VAR_INST
    {attribute 'hide'}
    bEncError           : BOOL;
END_VAR
// Save Encoder position
// needs some pre-conditions to use persistent storage
IF Enable THEN
    // Check ST_MotionStage for an encoder error (range 0x44nn)
    bEncError:=  stMotionStage.Axis.Status.Error AND  (  stMotionStage.Axis.Status.ErrorID  >= 16#4400  AND  stMotionStage.Axis.Status.ErrorID <= 16#44FF );
    // Do not save if we're currently loading or if there is an encoder error
    IF NOT bRestoreLoad AND NOT bEncError AND NOT bRestoreWaitRetry THEN
        fSavedPosition :=  stMotionStage.Axis.NcToPlc.ActPos;
        // This persistent variable lets us check if anything was saved
        // It will be TRUE at startup if we have saved values
        bSaved := TRUE;
    END_IF
END_IF
END_METHOD

{attribute 'call_after_init'}
(*  eModule: Mandatory must be unique for each MCS2 axis
    clears startup errors or warnings. the process is completed at run time
    SDO update of Drive and open Loop parameter Indexes based on module number
*)
METHOD PostInit
(* SDO update of Drive and open Loop parameter Indexes based on module number *)
stChanParams.nChanErrorCodeIdx        	:= nChanErrorCodeBase         	+ ((eModule-1) * nChanOfsBase);
stChanParams.nChanFErrWinIdx          	:= nChanFErrWinBase           	+ ((eModule-1) * nChanOfsBase);
stChanParams.nChanSoftLimitIdx        	:= nChanSoftLimitBase     		+ ((eModule-1) * nChanOfsBase);
stChanParams.nChanHomeOffsIdx         	:= nChanHomeOffsetBase        	+ ((eModule-1) * nChanOfsBase);
stChanParams.nChanHomeMethodIdx         := nChanHomeMethodBase       	+ ((eModule-1) * nChanOfsBase);
stChanParams.nChanHomeVeloIdx         	:= nChanHomingSpeedBase       	+ ((eModule-1) * nChanOfsBase);
stChanParams.nChanhomeAccIdx          	:= nChanhomingAccBase         	+ ((eModule-1) * nChanOfsBase);
stChanParams.nChanStepIdx             	:= nChanOlStepBase            	+ ((eModule-1) * nChanOfsBase);
stChanParams.nChanStepFreqIdx         	:= nChanOlStepFreqBase        	+ ((eModule-1) * nChanOfsBase);
stChanParams.nChanStepAmpIdx          	:= nChanOlStepAmpBase         	+ ((eModule-1) * nChanOfsBase);
stChanParams.nChanMaxCloseLoopFreqIdx   := nChanMaxCloseLoopFreqBase  	+ ((eModule-1) * nChanOfsBase);
stChanParams.nChanPositionerTypeIdx     := nChanPositionerTypeBase    	+ ((eModule-1) * nChanOfsBase);
stChanParams.nChanCalibrationOptIdx     := nCHanCalibrationOptBase    	+ ((eModule-1) * nChanOfsBase);
stChanParams.nChanSensorPowerModeIdx    := nChanSensorPowerModeBase   	+ ((eModule-1) * nChanOfsBase);
stChanParams.nChanReferencingOptIdx     := nChanReferencingOptBase    	+ ((eModule-1) * nChanOfsBase);
stChanParams.nChanReferenceTypeIdx      := nChanReferenceTypeBase     	+ ((eModule-1) * nChanOfsBase);
stChanParams.nChanSafeDirIdx            := nChanSafeDirBase           	+ ((eModule-1) * nChanOfsBase);
stChanParams.nChanMotorLoadIdx          := nChanMotorLoadBase         	+ ((eModule-1) * nChanOfsBase);
stChanParams.nChannelTypeIdx          	:= nChannelTypeBase       		+ ((eModule-1) * nChanOfsBase);
stChanParams.nChanStateIdx         		:= nChannelStateBase      		+ ((eModule-1) * nChanOfsBase);
stChanParams.nChanLogicalScaleOfsIdx   	:= nChanLogicalScaleOffsetBase	+ ((eModule-1) * nChanOfsBase);
stChanParams.nChanLogicalScaleInvIdx    := nChanLogicalScaleInvBase   	+ ((eModule-1) * nChanOfsBase);
stChanParams.nChanChannelTempIdx        := nChanChannelTempBase       	+ ((eModule-1) * nChanOfsBase);
stChanParams.nChanMovementTypeIdx       := nChanMovementTypeBase      	+ ((eModule-1) * nChanOfsBase);
stChanParams.nChanBaseUnitIdx           := nChanBaseUnitBase          	+ ((eModule-1) * nChanOfsBase);
stChanParams.nChanBaseResolutionIdx     := nChanBaseResolutionBase    	+ ((eModule-1) * nChanOfsBase);
stChanParams.nChanDistCodeInvIdx        := nChanDistCodeInvBase       	+ ((eModule-1) * nChanOfsBase);
stChanParams.nChanPositionerCtrlOptIdx  := nChanPositionerCtrlOptBase 	+ ((eModule-1) * nChanOfsBase);
stChanParams.nChanActuatorModeIdx       := nChanActuatorModeBase      	+ ((eModule-1) * nChanOfsBase);
stChanParams.nChanMotorLoadProtIdx      := nChanMotorLoadProtBase     	+ ((eModule-1) * nChanOfsBase);
stChanParams.nChanDiagClfIdx            := nChanDiagClfBase           	+ ((eModule-1) * nChanOfsBase);
bSystemInit := TRUE;
END_METHOD

METHOD PRIVATE PostMoveChecks : BOOL
VAR_INST
    rtAbortedHome        : R_TRIG;
    rtAbortedStepMove    : R_TRIG;
    rtAbortedCalibration : R_TRIG;
    rtResetDone          : R_TRIG;
    rtHaltDone           : R_TRIG;
    rtMoveDone           : R_TRIG;
    rtHomeDone           : R_TRIG;
    rtStepMoveDone       : R_TRIG;
    rtCalibrationDone    : R_TRIG;
    ftEnableFallEdge     : F_TRIG;
END_VAR
rtAbortedHome(CLK := fbhome.bHomeMoveAborted);
rtAbortedStepMove(CLK := fbStepMode.bStepMoveAborted);
rtAbortedCalibration(CLK := fbCalibrate.bCalibrateMoveAborted);

rtResetDone(CLK := fbMcReset.Done);
rtHaltDone(CLK := fbMcHalt.Done);

rtMoveDone(CLK := fbMcMoveAbsolute.Done);
rtHomeDone(CLK := fbhome.bHomeMoveDone);
rtStepMoveDone(CLK := fbStepMode.bStepMoveDone);
rtCalibrationDone(CLK := fbCalibrate.bCalibrateMoveDone);

IF rtAbortedHome.Q OR rtAbortedStepMove.Q OR rtAbortedCalibration.Q
   OR rtResetDone.Q OR rtHaltDone.Q
   OR rtMoveDone.Q OR rtHomeDone.Q OR rtStepMoveDone.Q OR rtCalibrationDone.Q THEN

    IF NOT stMotionStage.bDone THEN
        stMotionStage.bExecute := FALSE;;
        stMotionStage.bHomed := fbhome.bHomeMoveDone;
        IF rtMoveDone.Q THEN
            stMotionStage.bDone := TRUE;
            eDoneCause := E_MoveDoneCause.MoveDone;
        ELSIF rtStepMoveDone.Q THEN
            stMotionStage.bDone := TRUE;
            eDoneCause := E_MoveDoneCause.StepMoveDone;
        ELSIF rtHomeDone.Q THEN
            stMotionStage.bDone := TRUE;
            eDoneCause := E_MoveDoneCause.HomeDone;
            // Homing runs in DS402 manual HOME mode. Request closed-loop so the
            // drive manager switches the drive back to CSP now that homing is done.
            stChanParams.eOpModeReq := E_MCS2OpModeReq.CLOSED_LOOP;
        ELSIF rtCalibrationDone.Q THEN
            stMotionStage.bDone := TRUE;
            eDoneCause := E_MoveDoneCause.CalibrationDone;
            // Calibration runs in DS402 manual CALIBRATE mode. Request closed-loop so
            // the drive manager switches the drive back to CSP now that calibration is done.
            stChanParams.eOpModeReq := E_MCS2OpModeReq.CLOSED_LOOP;
        ELSIF rtResetDone.Q THEN
            stMotionStage.bDone := TRUE;
            eDoneCause := E_MoveDoneCause.ResetDone;
        ELSIF rtHaltDone.Q THEN
            stMotionStage.bDone := TRUE;
            eDoneCause := E_MoveDoneCause.HaltDone;
        ELSIF rtAbortedHome.Q THEN
            stMotionStage.bDone := TRUE;
            eDoneCause := E_MoveDoneCause.AbortedHome;
        ELSIF rtAbortedStepMove.Q THEN
            stMotionStage.bDone := TRUE;
            eDoneCause := E_MoveDoneCause.AbortedStepMove;
        ELSIF rtAbortedCalibration.Q THEN
            stMotionStage.bDone := TRUE;
            eDoneCause := E_MoveDoneCause.AbortedCalibration;
        END_IF
        IF rtHomeDone.Q OR rtAbortedHome.Q OR rtCalibrationDone.Q OR rtAbortedCalibration.Q THEN
            bEnPosLag       := bRecentEnPosLagStatus;
            fParameterValue := BOOL_TO_LREAL(bRecentEnPosLagStatus);
        END_IF
        IF fbDriveManager.bDS402Manual
           AND NOT (rtHomeDone.Q OR rtAbortedHome.Q OR rtCalibrationDone.Q OR rtAbortedCalibration.Q) THEN
            bEnPosLag := FALSE;
        END_IF
        IF (stMotionStage.nEnableMode = E_StageEnableMode.DURING_MOTION) THEN
            bPositionHold := TRUE;
            tonHoldTime.IN := TRUE;
        END_IF
        // get stable current position storage
        stChanParams.fPosition := stMotionStage.fPosition;
    END_IF
END_IF

tonHoldTime(PT := UDINT_TO_TIME(stChanParams.nHoldTime));
IF tonHoldTime.Q THEN
    bPositionHold := FALSE;
    tonHoldTime.IN := FALSE;
    bLastHoltTimeOut := TRUE;
END_IF

(* updated axis status
   Not needed in manual mode *)
IF NOT fbDriveManager.bDS402Manual THEN
     stMotionStage.Axis.ReadStatus();
END_IF

bPrepareDisable S= (stMotionStage.nEnableMode = E_StageEnableMode.DURING_MOTION) AND ftExec.Q;

IF bPrepareDisable AND fbDriveManager.bCSPModeEnabled THEN
    IF stMotionStage.Axis.Status.StandStill THEN
        IF NOT bPositionHold THEN
            bPrepareDisable := FALSE;
            stMotionStage.bEnable := FALSE; // TwinCAT NC disables MC_Power (CSP)
        END_IF
    END_IF
ELSIF bPrepareDisable AND fbDriveManager.bDS402Manual THEN
    IF fbDriveManager.bOperational THEN
        IF NOT bPositionHold THEN
            bPrepareDisable := FALSE;
            stMotionStage.bEnable := FALSE; // Manual disables via drive control word
        END_IF
    END_IF
END_IF

ftEnableFallEdge(CLK := stMotionStage.bEnable);
IF ftEnableFallEdge.Q THEN
    // Only power off in manual if we're staying in manual. During a switch back
    // to CSP, let the NC ramp the control word down so it isn't disabled under it.
    IF fbDriveManager.bDS402Manual
       AND stChanParams.eOpModeReq <> E_MCS2OpModeReq.CLOSED_LOOP THEN
        stDS402Drive.nDriveControl := 6; // Manual mode power off
    END_IF
END_IF
END_METHOD

METHOD Power
fbMcPower(
    Axis :=  stMotionStage.Axis,
    Enable :=  stMotionStage.bAllEnable,
    Enable_Positive :=  stMotionStage.bAllForwardEnable AND stChanParams.bOverrideDirEnable,
    Enable_Negative :=  stMotionStage.bAllBackwardEnable AND stChanParams.bOverrideDirEnable,
    Override := 100.0,
    BufferMode := MC_BufferMode.MC_Aborting
);
END_METHOD

METHOD Reset
fbMcReset(
    Axis :=  stMotionStage.Axis,
    Execute := bReset
);
IF fbMcReset.Done THEN
    bReset := FALSE;
END_IF
END_METHOD

METHOD RestoreMotionParams
VAR_INPUT
    Enable  : BOOL;
END_VAR

VAR_INST
    fbSetPos            : MC_SetPosition;
    {attribute 'hide'}
    bLoad               : BOOL;
    {attribute 'hide'}
    bRestoreInit        : BOOL;
    {attribute 'hide'}
    nMaxRetries         : UINT := 10;
    {attribute 'hide'}
    nCurrTries          : UINT := 0;
    {attribute 'hide'}
    nLatchError         : UDINT;
END_VAR
IF Enable THEN
    // Trigger a load if anything was saved at all
    IF NOT bRestoreInit THEN
        bRestoreInit := TRUE;
        bRestoreLoad S= bSaved;
        fbSetPos.Options.ClearPositionLag := TRUE;
    END_IF

    // Set our position if bRestoreLoad is true
    fbSetPos( Axis:= stMotionStage.Axis, Execute:=bRestoreLoad, Position:=fSavedPosition);

    IF fbSetPos.Error THEN
        // Keep the error latched, it can disappear if Execute is set to FALSE
        nLatchError := fbSetPos.ErrorID;
        nCurrTries := nCurrTries + 1;
        IF nCurrTries >= nMaxRetries THEN
        // Alert the user that something has gone wrong
         stMotionStage.bError := TRUE;
         stMotionStage.nErrorId := nLatchError;
         stMotionStage.sCustomErrorMessage := 'Error loading previously saved position.';
        ELSE
            // Reset the FB for the next retry
            fbSetPos( Axis:= stMotionStage.Axis, Execute:=bRestoreLoad, Position:=fSavedPosition);
            // Try again
            bRestoreWaitRetry := TRUE;
        END_IF
    ELSIF fbSetPos.Done THEN
         stMotionStage.fPosition := fSavedPosition;
         stMotionStage.bRestoreDone := TRUE;
    END_IF

    // Only load once, at startup
    bRestoreLoad R= fbSetPos.Done OR fbSetPos.Error;

    tonRestoreRetry( IN := bRestoreWaitRetry, PT := T#100MS);
    bRestoreLoad S= tonRestoreRetry.Q;
    bRestoreWaitRetry R= tonRestoreRetry.Q;
END_IF
END_METHOD

METHOD ScaleEncRawValue
VAR_INPUT
  //  bEnable: BOOL;
END_VAR
(* SmartACT: The encoder count from the Piezo drive is not a raw count from the embeded actuator device
   we get a calibrated nm value. thus the use of abs() since this value is signed.*)

stMotionStage.nEncoderCount:=DINT_TO_UDINT(ABS( stMotionStage.nRawEncoderDINT));

// calibrated encoder readback
IF NOT fbDriveManager.bStepModeEnabled THEN
    // Close loop NC
    fMeasuredPos:= stMotionStage.Axis.NcToPlc.ActPos;
    fMeasuredVelo := stMotionStage.Axis.NcToPlc.ActVelo;
    fMeasuredAcc :=  stMotionStage.Axis.NcToPlc.ActAcc;
    stMotionStage.fPosDiff:= stMotionStage.Axis.NcToPlc.PosDiff;
ELSE
    fMeasuredPos:=DINT_TO_REAL( stMotionStage.nRawEncoderDINT) * MAX( stMotionStage.stAxisParameters.fEncScaleFactorInternal, stChanParams.fScalingFactor);
    stMotionStage.fPosDiff:= stMotionStage.fPosition - fMeasuredPos;
    // NB: Not actual in open loop
    fMeasuredVelo := stMotionStage.fVelocity;
    fMeasuredAcc :=  stMotionStage.fAcceleration;
END_IF
END_METHOD

METHOD SetEnables
VAR_INPUT
END_VAR
 stMotionStage.bAllForwardEnable:= stMotionStage.bLimitForwardEnable
                                    AND ( stMotionStage.bGantryForwardEnable OR NOT  stMotionStage.bGantryAxis)
                                    AND  stMotionStage.stEPSForwardEnable.bEPS_OK
                                    AND  stChanParams.bOverrideDirEnable;
 stMotionStage.bAllBackwardEnable:= stMotionStage.bLimitBackwardEnable
                                    AND ( stMotionStage.bGantryBackwardEnable OR NOT  stMotionStage.bGantryAxis)
                                    AND  stMotionStage.stEPSBackwardEnable.bEPS_OK
                                    AND  stChanParams.bOverrideDirEnable;

 stMotionStage.bAllEnable:= stMotionStage.bEnable
                            AND  stMotionStage.bHardwareEnable
                            AND  stMotionStage.stEPSPowerEnable.bEPS_OK;
 stMotionStage.bAllEnable R= NOT  stMotionStage.bUserEnable;
END_METHOD

METHOD UpdateEpicsStatus
VAR_INPUT
END_VAR
//////////////////////////////////////////////////////////////////
// Transfer NC parameter status to EPICS
//////////////////////////////////////////////////////////////////
 stMotionStage.nMotionAxisID :=  stMotionStage.Axis.NcToPlc.AxisId;
 stMotionStage.stAxisStatus.bEnable:= stMotionStage.bAllEnable;
 stMotionStage.stAxisStatus.bEnabled:= stMotionStage.bEnableDone; // account for PowerEnable from power block
 stMotionStage.stAxisStatus.bError:= stMotionStage.bError;
 stMotionStage.stAxisStatus.bHomeSensor:= stMotionStage.bHome;
 stMotionStage.stAxisStatus.bLimitBwd:= stMotionStage.bAllBackwardEnable;
 stMotionStage.stAxisStatus.bLimitFwd:= stMotionStage.bAllForwardEnable;
 stMotionStage.stAxisStatus.bReset:= stMotionStage.bReset;
 stMotionStage.stAxisStatus.fAcceleration:=fMeasuredAcc;
 stMotionStage.stAxisStatus.fActDiff:= stMotionStage.fPosDiff;
 stMotionStage.stAxisStatus.fActPosition:=fMeasuredPos;
 stMotionStage.stAxisStatus.fActVelocity:=fMeasuredVelo;
 stMotionStage.stAxisStatus.fDeceleration:=fMeasuredAcc;
 stMotionStage.stAxisStatus.fOverride:=fbMcPower.Override;
 stMotionStage.stAxisStatus.fPosition:= stMotionStage.fPosition;
 stMotionStage.stAxisStatus.fVelocity:= stMotionStage.fVelocity;
 stMotionStage.stAxisStatus.nCmdData:=INT_TO_UINT( stMotionStage.nCmdData);  //Or nCmdDataLocal
 stMotionStage.stAxisStatus.nCommand:=INT_TO_UINT( stMotionStage.nCommand);  //Or nCommandLocal
 stMotionStage.stAxisStatus.nErrorId:= stMotionStage.nErrorId;
 stMotionStage.stAxisStatus.bBusy:= stMotionStage.bBusy;
 stMotionStage.stAxisStatus.bHomed:= stMotionStage.bHomed;
 stMotionStage.stAxisStatus.bExecute:=bLocalExec;
 stMotionStage.stAxisStatus.nCommand:=3; // If this is not 3, the IOC stops updating positions during homing
END_METHOD

METHOD WriteParameterNC
VAR_INPUT
    Execute:BOOL;
    ParameterNumber : MC_AxisParameter;
    ParameterValue  : LREAL;
END_VAR
(*Do not change a moving axis parameter*)
fbMcWriteParameter(
    Axis:=stMotionStage.Axis,
    Execute:=(Execute AND stMotionStage.Axis.Status.NotMoving),
    ParameterNumber:=ParameterNumber,
    Value:=ParameterValue
);
END_METHOD

END_FUNCTION_BLOCK

// ---- POUs/Motion/DS402/MCS2/FB_WriteChanParameters.TcPOU
// Consolidated SDO parameter writer for MCS2 drives.
//
// At boot: every SDO write runs once in a single sequential FSM. The CoE
// mailbox sees one outstanding write at a time, eliminating the random
// boot-time failures caused by overlapping requests.
//
// After boot: each parameter is monitored independently and written in
// parallel/on-demand when its setpoint changes (operator/EPICS edits).
//
// Drive an error reset via bErrorAcknowledge to restart the sequence.

FUNCTION_BLOCK FB_WriteChanParameters
VAR_INPUT
    bEnable             : BOOL;
    bErrorAcknowledge   : BOOL;
    // Debug: force the full sequential sweep to re-run.
    bForceSequentialSDOs : BOOL := FALSE;
END_VAR

VAR_IN_OUT
    stDS402Drive        : ST_DS402Drive;
    stMotionStage       : ST_MotionStage;
    stChanParams 		: ST_MCS2ChanParameter;
END_VAR

VAR_OUTPUT
    bParamsSet : BOOL;
END_VAR

VAR
    // Channel parameters
    fbSetFErrorWin            : FB_EcCoESdoWrite;
    fbSetSoftLimMin           : FB_EcCoESdoWrite;
    fbSetSoftLimMax           : FB_EcCoESdoWrite;
    fbMaxCloseLoopFreqWrite   : FB_EcCoESdoWrite;
    fbSensorPowerModeWrite    : FB_EcCoESdoWrite;
    fbLogicalScaleOffsetWrite : FB_EcCoESdoWrite;
    fbLogicalScaleInvWrite    : FB_EcCoESdoWrite;
    fbSafeDirWrite            : FB_EcCoESdoWrite;
    fbDistCodeInvWrite        : FB_EcCoESdoWrite;
    fbPositionerCtrlOptWrite  : FB_EcCoESdoWrite;
    fbActuatorModeWrite       : FB_EcCoESdoWrite;
    fbMotorLoadProtWrite      : FB_EcCoESdoWrite;
    // Calibration parameters
    fbCalibrationOptWrite     : FB_EcCoESdoWrite;
    // Home parameters
    fbSetHomeVeloFast         : FB_EcCoESdoWrite;
    fbSetHomeVeloSlow         : FB_EcCoESdoWrite;
    fbSetHomeAcc              : FB_EcCoESdoWrite;
    fbSetHomeOffs             : FB_EcCoESdoWrite;
    fbSetHomeMethod             : FB_EcCoESdoWrite;
    fbReferencingOptWrite     : FB_EcCoESdoWrite;
    // Step-mode parameters
    fbSetSteps                : FB_EcCoESdoWrite;
    fbSetStepAmp              : FB_EcCoESdoWrite;
    fbSetStepFreq             : FB_EcCoESdoWrite;

    // Channel
    {attribute 'hide'}
    nRecentFErrWin              : DINT;
    {attribute 'hide'}
    nRecentSoftLimMin           : LINT;
    {attribute 'hide'}
    nRecentSoftLimMax           : LINT;
    {attribute 'hide'}
    nRecentMaxCloseLoopFreq     : UDINT;
    {attribute 'hide'}
    nRecentSensorPowerMode      : UDINT;
    {attribute 'hide'}
    nRecentLogicalScaleOffset   : LINT;
    {attribute 'hide'}
    nRecentLogicalScaleInv      : BOOL;
    {attribute 'hide'}
    nRecentSafeDir              : BOOL;
    {attribute 'hide'}
    nRecentDistCodeInv          : BOOL;
    {attribute 'hide'}
    nRecentPositionerCtrlOpt    : DWORD;
    {attribute 'hide'}
    nRecentActuatorMode         : UDINT;
    {attribute 'hide'}
    nRecentMotorLoadProt        : USINT;

    // Calibration
    {attribute 'hide'}
    nRecentCalibrationOpt       : UDINT;
    // Home
    {attribute 'hide'}
    nRecentHomeVeloFast         : UDINT;
    {attribute 'hide'}
    nRecentHomeVeloSlow         : UDINT;
    {attribute 'hide'}
    nRecentHomeAcc              : UDINT;
    {attribute 'hide'}
    nRecentHomeOffset           : DINT;
    {attribute 'hide'}
    nRecentHomeMethod			: SINT;
    {attribute 'hide'}
    nRecentReferencingOpt       : UDINT;
    // Step-mode
    {attribute 'hide'}
    nRecentSteps                : DINT;
    {attribute 'hide'}
    nRecentStepAmp              : UINT;
    {attribute 'hide'}
    nRecentStepFreq             : UINT;

    {attribute 'hide'}
    ftFErrWinSetDone            : F_TRIG;
    {attribute 'hide'}
    ftSoftLimMinSetDone         : F_TRIG;
    {attribute 'hide'}
    ftSoftLimMaxSetDone         : F_TRIG;
    {attribute 'hide'}
    ftMaxCloseLoopFreqSetDone   : F_TRIG;
    {attribute 'hide'}
    ftSensorPowerModeSetDone    : F_TRIG;
    {attribute 'hide'}
    ftLogicalScaleOffsetSetDone : F_TRIG;
    {attribute 'hide'}
    ftLogicalScaleInvSetDone    : F_TRIG;
    {attribute 'hide'}
    ftSafeDirSetDone            : F_TRIG;
    {attribute 'hide'}
    ftDistCodeInvSetDone        : F_TRIG;
    {attribute 'hide'}
    ftPositionerCtrlOptSetDone  : F_TRIG;
    {attribute 'hide'}
    ftActuatorModeSetDone       : F_TRIG;
    {attribute 'hide'}
    ftMotorLoadProtSetDone      : F_TRIG;
    {attribute 'hide'}
    ftCalibrationOptSetDone     : F_TRIG;
    {attribute 'hide'}
    ftHomeVeloFastSetDone       : F_TRIG;
    {attribute 'hide'}
    ftHomeVeloSlowSetDone       : F_TRIG;
    {attribute 'hide'}
    ftHomeAccSetDone            : F_TRIG;
    {attribute 'hide'}
    ftHomeOffsSetDone           : F_TRIG;
    {attribute 'hide'}
    ftHomeMethodSetDone         : F_TRIG;
    {attribute 'hide'}
    ftReferencingOptSetDone     : F_TRIG;
    {attribute 'hide'}
    ftStepUpdateDone            : F_TRIG;
    {attribute 'hide'}
    ftStepAmpUpdateDone         : F_TRIG;
    {attribute 'hide'}
    ftStepFreqUpdateDone        : F_TRIG;

    // Scaled / derived parameter values
    nScaledFErrWin    : DINT;
    nScalededSteps    : DINT;
    nScalededStepAmp  : UINT;
    nScaledStepFreq   : UINT;

    // Boot-time one-shot sequential FSM

    // tonInitialDelay only gates the *first* sweep after enable.
    tonInitialDelay : TON;
    bSweepArmed     : BOOL;
    bSweepActive    : BOOL;
    bBootSweepDone  : BOOL;
    // TRUE while the linked EtherCAT slave is in PreOp ESM state.
    {attribute 'hide'}
    bInPreOp        : BOOL;
    eBootStep : (
        IDLE     := 0,
        // Channel
        FERR     := 1,
        SOFTMIN  := 2,
        SOFTMAX  := 3,
        CLOSEFREQ:= 4,
        SENSORPWR:= 5,
        SCALEOFS := 6,
        SCALEINV := 7,
        // Calibration
        CALIBOPT := 8,
        // Home
        HOME_VELO_FAST := 9,
        HOME_VELO_SLOW := 10,
        HOME_ACC       := 11,
        HOME_OFFSET    := 12,
        HOME_METHOD    := 13,
        HOME_REF_OPT   := 14,
        // Step-mode
        STEPS    := 15,
        STEP_AMP := 16,
        STEP_FREQ:= 17,
        // Extra channel params
        DIST_CODE_INV   := 18,
        POS_CTRL_OPT    := 19,
        ACT_MODE        := 20,
        MOTOR_LOAD_PROT := 21,
        SAFEDIR         := 22,
        DONE     := 100,
        ERR      := -1
    ) := IDLE;
END_VAR

IF NOT __ISVALIDREF(stDS402Drive)
    OR NOT __ISVALIDREF(stMotionStage)
    OR NOT __ISVALIDREF(stChanParams) THEN
    RETURN;
END_IF

IF NOT bEnable THEN
    RETURN;
END_IF

// Logical Scale Inversion (0x2009) and Safe Direction (0x200C) are writable
// only in PreOp ESM state. Gate their writes on the linked slave state so an
// OP-state write cannot raise a runtime SDO error. The low nibble of
// InfoData.State is the ESM state (2=PreOp).
bInPreOp := (stDS402Drive.nEcatState AND 16#000F) = 2;

// Initial boot delay: only used to arm the first sweep.
tonInitialDelay(
    IN := bEnable AND NOT bSweepArmed,
    PT := stChanParams.nReadTime
);
IF tonInitialDelay.Q THEN
    bSweepArmed := TRUE;
END_IF

// Error acknowledge restarts the sweep without re-paying the 6 s delay.
IF eBootStep = ERR AND bErrorAcknowledge THEN
    eBootStep              := IDLE;
    bBootSweepDone         := FALSE;
    bSweepActive           := TRUE;
END_IF

// Force a re-sweep on demand.
IF bForceSequentialSDOs THEN
    bBootSweepDone := FALSE;
    bSweepActive   := TRUE;
    eBootStep      := IDLE;
END_IF

// Arm the first sweep when the initial delay completes.
IF bSweepArmed AND NOT bBootSweepDone AND NOT bSweepActive THEN
    bSweepActive := TRUE;
    eBootStep    := IDLE;
END_IF

// Pre-compute scaled values every cycle.
ScaleDriveParams();
ScaleHomingParams();
ScaleStepModeParams();

// Drive falling-edge detectors (one shared block for both modes).
ftFErrWinSetDone           (CLK := fbSetFErrorWin.bBusy);
ftSoftLimMinSetDone        (CLK := fbSetSoftLimMin.bBusy);
ftSoftLimMaxSetDone        (CLK := fbSetSoftLimMax.bBusy);
ftMaxCloseLoopFreqSetDone  (CLK := fbMaxCloseLoopFreqWrite.bBusy);
ftSensorPowerModeSetDone   (CLK := fbSensorPowerModeWrite.bBusy);
ftLogicalScaleOffsetSetDone(CLK := fbLogicalScaleOffsetWrite.bBusy);
ftLogicalScaleInvSetDone   (CLK := fbLogicalScaleInvWrite.bBusy);
ftSafeDirSetDone           (CLK := fbSafeDirWrite.bBusy);
ftDistCodeInvSetDone       (CLK := fbDistCodeInvWrite.bBusy);
ftPositionerCtrlOptSetDone (CLK := fbPositionerCtrlOptWrite.bBusy);
ftActuatorModeSetDone      (CLK := fbActuatorModeWrite.bBusy);
ftMotorLoadProtSetDone     (CLK := fbMotorLoadProtWrite.bBusy);
ftCalibrationOptSetDone    (CLK := fbCalibrationOptWrite.bBusy);
ftHomeVeloFastSetDone      (CLK := fbSetHomeVeloFast.bBusy);
ftHomeVeloSlowSetDone      (CLK := fbSetHomeVeloSlow.bBusy);
ftHomeAccSetDone           (CLK := fbSetHomeAcc.bBusy);
ftHomeOffsSetDone          (CLK := fbSetHomeOffs.bBusy);
ftHomeMethodSetDone        (CLK := fbSetHomeMethod.bBusy);
ftReferencingOptSetDone    (CLK := fbReferencingOptWrite.bBusy);
ftStepUpdateDone           (CLK := fbSetSteps.bBusy);
ftStepAmpUpdateDone        (CLK := fbSetStepAmp.bBusy);
ftStepFreqUpdateDone       (CLK := fbSetStepFreq.bBusy);

IF bSweepActive THEN
    bParamsSet := FALSE;
    BootSweepStep();
ELSIF eBootStep = ERR THEN
    HoldAllWritersIdle();
ELSIF bBootSweepDone THEN
    ParallelOnDemand();
ELSE
    // Pre-boot: keep every writer fully idle.
    HoldAllWritersIdle();
END_IF

CallAllSdoWriters();

// After the boot sweep, bParamsSet reflects writer activity in real time:
// TRUE when no parameter writer is busy, FALSE while any is busy. The
IF bBootSweepDone THEN
    bParamsSet := NOT (
        fbSetFErrorWin.bBusy
        OR fbSetSoftLimMin.bBusy
        OR fbSetSoftLimMax.bBusy
        OR fbMaxCloseLoopFreqWrite.bBusy
        OR fbSensorPowerModeWrite.bBusy
        OR fbLogicalScaleOffsetWrite.bBusy
        OR fbLogicalScaleInvWrite.bBusy
        OR fbSafeDirWrite.bBusy
        OR fbCalibrationOptWrite.bBusy
        OR fbSetHomeVeloFast.bBusy
        OR fbSetHomeVeloSlow.bBusy
        OR fbSetHomeAcc.bBusy
        OR fbSetHomeOffs.bBusy
        OR fbSetHomeMethod.bBusy
        OR fbReferencingOptWrite.bBusy
        OR fbSetSteps.bBusy
        OR fbSetStepAmp.bBusy
        OR fbSetStepFreq.bBusy
        OR fbDistCodeInvWrite.bBusy
        OR fbPositionerCtrlOptWrite.bBusy
        OR fbActuatorModeWrite.bBusy
        OR fbMotorLoadProtWrite.bBusy
    );
END_IF

// One step of the boot-time sequential sweep.
// Pattern per step: if value matches cache, skip; otherwise execute the SDO
// write and wait for its busy->idle falling edge before advancing.
METHOD PRIVATE BootSweepStep
CASE eBootStep OF

    IDLE:
        // Clear every execute line at start of sweep so nothing carries over.
        fbSetFErrorWin.bExecute            := FALSE;
        fbSetSoftLimMin.bExecute           := FALSE;
        fbSetSoftLimMax.bExecute           := FALSE;
        fbMaxCloseLoopFreqWrite.bExecute   := FALSE;
        fbSensorPowerModeWrite.bExecute    := FALSE;
        fbLogicalScaleOffsetWrite.bExecute := FALSE;
        fbLogicalScaleInvWrite.bExecute    := FALSE;
        fbSafeDirWrite.bExecute            := FALSE;
        fbCalibrationOptWrite.bExecute     := FALSE;
        fbSetHomeVeloFast.bExecute         := FALSE;
        fbSetHomeVeloSlow.bExecute         := FALSE;
        fbSetHomeAcc.bExecute              := FALSE;
        fbSetHomeOffs.bExecute             := FALSE;
        fbSetHomeMethod.bExecute           := FALSE;
        fbReferencingOptWrite.bExecute     := FALSE;
        fbSetSteps.bExecute                := FALSE;
        fbSetStepAmp.bExecute              := FALSE;
        fbSetStepFreq.bExecute             := FALSE;
        fbDistCodeInvWrite.bExecute        := FALSE;
        fbPositionerCtrlOptWrite.bExecute  := FALSE;
        fbActuatorModeWrite.bExecute       := FALSE;
        fbMotorLoadProtWrite.bExecute      := FALSE;
        eBootStep := FERR;

    // Channel params
    FERR:
        IF nScaledFErrWin <> nRecentFErrWin THEN
            fbSetFErrorWin.bExecute := TRUE;
            IF ftFErrWinSetDone.Q THEN
                fbSetFErrorWin.bExecute := FALSE;
                IF fbSetFErrorWin.bError THEN
                    stMotionStage.bError   := fbSetFErrorWin.bError;
                    stMotionStage.nErrorId := fbSetFErrorWin.nErrId;
                    eBootStep              := ERR;
                ELSE
                    nRecentFErrWin := nScaledFErrWin;
                    eBootStep      := SOFTMIN;
                END_IF
            END_IF
        ELSE
            eBootStep := SOFTMIN;
        END_IF

    SOFTMIN:
        IF stChanParams.nSoftLimMin <> nRecentSoftLimMin THEN
            fbSetSoftLimMin.bExecute := TRUE;
            IF ftSoftLimMinSetDone.Q THEN
                fbSetSoftLimMin.bExecute := FALSE;
                IF fbSetSoftLimMin.bError THEN
                    stMotionStage.bError   := fbSetSoftLimMin.bError;
                    stMotionStage.nErrorId := fbSetSoftLimMin.nErrId;
                    eBootStep              := ERR;
                ELSE
                    nRecentSoftLimMin := stChanParams.nSoftLimMin;
                    eBootStep         := SOFTMAX;
                END_IF
            END_IF
        ELSE
            eBootStep := SOFTMAX;
        END_IF

    SOFTMAX:
        IF stChanParams.nSoftLimMax <> nRecentSoftLimMax THEN
            fbSetSoftLimMax.bExecute := TRUE;
            IF ftSoftLimMaxSetDone.Q THEN
                fbSetSoftLimMax.bExecute := FALSE;
                IF fbSetSoftLimMax.bError THEN
                    stMotionStage.bError   := fbSetSoftLimMax.bError;
                    stMotionStage.nErrorId := fbSetSoftLimMax.nErrId;
                    eBootStep              := ERR;
                ELSE
                    nRecentSoftLimMax := stChanParams.nSoftLimMax;
                    eBootStep         := CLOSEFREQ;
                END_IF
            END_IF
        ELSE
            eBootStep := CLOSEFREQ;
        END_IF

    CLOSEFREQ:
        IF stChanParams.nMaxCloseLoopFreq <> nRecentMaxCloseLoopFreq THEN
            fbMaxCloseLoopFreqWrite.bExecute := TRUE;
            IF ftMaxCloseLoopFreqSetDone.Q THEN
                fbMaxCloseLoopFreqWrite.bExecute := FALSE;
                IF fbMaxCloseLoopFreqWrite.bError THEN
                    stMotionStage.bError   := fbMaxCloseLoopFreqWrite.bError;
                    stMotionStage.nErrorId := fbMaxCloseLoopFreqWrite.nErrId;
                    eBootStep              := ERR;
                ELSE
                    nRecentMaxCloseLoopFreq := stChanParams.nMaxCloseLoopFreq;
                    eBootStep               := SENSORPWR;
                END_IF
            END_IF
        ELSE
            eBootStep := SENSORPWR;
        END_IF

    SENSORPWR:
        IF stChanParams.nSensorPowerMode <> nRecentSensorPowerMode THEN
            fbSensorPowerModeWrite.bExecute := TRUE;
            IF ftSensorPowerModeSetDone.Q THEN
                fbSensorPowerModeWrite.bExecute := FALSE;
                IF fbSensorPowerModeWrite.bError THEN
                    stMotionStage.bError   := fbSensorPowerModeWrite.bError;
                    stMotionStage.nErrorId := fbSensorPowerModeWrite.nErrId;
                    eBootStep              := ERR;
                ELSE
                    nRecentSensorPowerMode := stChanParams.nSensorPowerMode;
                    eBootStep              := SCALEOFS;
                END_IF
            END_IF
        ELSE
            eBootStep := SCALEOFS;
        END_IF

    SCALEOFS:
        IF stChanParams.nLogicalScaleOffset <> nRecentLogicalScaleOffset THEN
            fbLogicalScaleOffsetWrite.bExecute := TRUE;
            IF ftLogicalScaleOffsetSetDone.Q THEN
                fbLogicalScaleOffsetWrite.bExecute := FALSE;
                IF fbLogicalScaleOffsetWrite.bError THEN
                    stMotionStage.bError   := fbLogicalScaleOffsetWrite.bError;
                    stMotionStage.nErrorId := fbLogicalScaleOffsetWrite.nErrId;
                    eBootStep              := ERR;
                ELSE
                    nRecentLogicalScaleOffset := stChanParams.nLogicalScaleOffset;
                    eBootStep                 := SCALEINV;
                END_IF
            END_IF
        ELSE
            eBootStep := SCALEINV;
        END_IF

    SCALEINV:
        // 0x2009 is PreOp-only. Skip during the boot sweep (the slave is in OP
        // by then) and only write when the slave is deliberately in PreOp;
        // ParallelOnDemand applies it whenever the setpoint diverges in PreOp.
        IF bInPreOp AND stChanParams.nLogicalScaleInv <> nRecentLogicalScaleInv THEN
            fbLogicalScaleInvWrite.bExecute := TRUE;
            IF ftLogicalScaleInvSetDone.Q THEN
                fbLogicalScaleInvWrite.bExecute := FALSE;
                IF fbLogicalScaleInvWrite.bError THEN
                    stMotionStage.bError   := fbLogicalScaleInvWrite.bError;
                    stMotionStage.nErrorId := fbLogicalScaleInvWrite.nErrId;
                    eBootStep              := ERR;
                ELSE
                    nRecentLogicalScaleInv := stChanParams.nLogicalScaleInv;
                    eBootStep              := SAFEDIR;
                END_IF
            END_IF
        ELSE
            eBootStep := SAFEDIR;
        END_IF

    SAFEDIR:
        // 0x200C is PreOp-only, same as 0x2009. Skip during the boot sweep (the
        // slave is in OP by then) and only write when the slave is deliberately
        // in PreOp; ParallelOnDemand applies it whenever the setpoint diverges.
        IF bInPreOp AND stChanParams.nSafeDir <> nRecentSafeDir THEN
            fbSafeDirWrite.bExecute := TRUE;
            IF ftSafeDirSetDone.Q THEN
                fbSafeDirWrite.bExecute := FALSE;
                IF fbSafeDirWrite.bError THEN
                    stMotionStage.bError   := fbSafeDirWrite.bError;
                    stMotionStage.nErrorId := fbSafeDirWrite.nErrId;
                    eBootStep              := ERR;
                ELSE
                    nRecentSafeDir := stChanParams.nSafeDir;
                    eBootStep      := CALIBOPT;
                END_IF
            END_IF
        ELSE
            eBootStep := CALIBOPT;
        END_IF

    // Calibration params
    CALIBOPT:
        IF stChanParams.nCalibrationOpt <> nRecentCalibrationOpt THEN
            fbCalibrationOptWrite.bExecute := TRUE;
            IF ftCalibrationOptSetDone.Q THEN
                fbCalibrationOptWrite.bExecute := FALSE;
                IF fbCalibrationOptWrite.bError THEN
                    stMotionStage.bError   := fbCalibrationOptWrite.bError;
                    stMotionStage.nErrorId := fbCalibrationOptWrite.nErrId;
                    eBootStep              := ERR;
                ELSE
                    nRecentCalibrationOpt := stChanParams.nCalibrationOpt;
                    eBootStep             := HOME_VELO_FAST;
                END_IF
            END_IF
        ELSE
            eBootStep := HOME_VELO_FAST;
        END_IF

    // Home params
    HOME_VELO_FAST:
        IF stChanParams.nHomeVeloFast <> nRecentHomeVeloFast THEN
            fbSetHomeVeloFast.bExecute := TRUE;
            IF ftHomeVeloFastSetDone.Q THEN
                fbSetHomeVeloFast.bExecute := FALSE;
                IF fbSetHomeVeloFast.bError THEN
                    stMotionStage.bError   := fbSetHomeVeloFast.bError;
                    stMotionStage.nErrorId := fbSetHomeVeloFast.nErrId;
                    eBootStep              := ERR;
                ELSE
                    nRecentHomeVeloFast := stChanParams.nHomeVeloFast;
                    eBootStep           := HOME_VELO_SLOW;
                END_IF
            END_IF
        ELSE
            eBootStep := HOME_VELO_SLOW;
        END_IF

    HOME_VELO_SLOW:
        IF stChanParams.nHomeVeloSlow <> nRecentHomeVeloSlow THEN
            fbSetHomeVeloSlow.bExecute := TRUE;
            IF ftHomeVeloSlowSetDone.Q THEN
                fbSetHomeVeloSlow.bExecute := FALSE;
                IF fbSetHomeVeloSlow.bError THEN
                    stMotionStage.bError   := fbSetHomeVeloSlow.bError;
                    stMotionStage.nErrorId := fbSetHomeVeloSlow.nErrId;
                    eBootStep              := ERR;
                ELSE
                    nRecentHomeVeloSlow := stChanParams.nHomeVeloSlow;
                    eBootStep           := HOME_ACC;
                END_IF
            END_IF
        ELSE
            eBootStep := HOME_ACC;
        END_IF

    HOME_ACC:
        IF stChanParams.nHomeAcc <> nRecentHomeAcc THEN
            fbSetHomeAcc.bExecute := TRUE;
            IF ftHomeAccSetDone.Q THEN
                fbSetHomeAcc.bExecute := FALSE;
                IF fbSetHomeAcc.bError THEN
                    stMotionStage.bError   := fbSetHomeAcc.bError;
                    stMotionStage.nErrorId := fbSetHomeAcc.nErrId;
                    eBootStep              := ERR;
                ELSE
                    nRecentHomeAcc := stChanParams.nHomeAcc;
                    eBootStep      := HOME_OFFSET;
                END_IF
            END_IF
        ELSE
            eBootStep := HOME_OFFSET;
        END_IF

    HOME_OFFSET:
        IF stChanParams.nHomeOffset <> nRecentHomeOffset THEN
            fbSetHomeOffs.bExecute := TRUE;
            IF ftHomeOffsSetDone.Q THEN
                fbSetHomeOffs.bExecute := FALSE;
                IF fbSetHomeOffs.bError THEN
                    stMotionStage.bError   := fbSetHomeOffs.bError;
                    stMotionStage.nErrorId := fbSetHomeOffs.nErrId;
                    eBootStep              := ERR;
                ELSE
                    nRecentHomeOffset := stChanParams.nHomeOffset;
                    eBootStep         := HOME_REF_OPT;
                END_IF
            END_IF
        ELSE
            eBootStep := HOME_METHOD;
        END_IF
    HOME_METHOD:
        IF stChanParams.nHomeMethod <> nRecentHomeMethod THEN
            fbSetHomeMethod.bExecute := TRUE;
            IF ftHomeMethodSetDone.Q THEN
                fbSetHomeMethod.bExecute := FALSE;
                IF fbSetHomeMethod.bError THEN
                    stMotionStage.bError   := fbSetHomeMethod.bError;
                    stMotionStage.nErrorId := fbSetHomeMethod.nErrId;
                    eBootStep              := ERR;
                ELSE
                    nRecentHomeMethod := stChanParams.nHomeMethod;
                    eBootStep         := HOME_REF_OPT;
                END_IF
            END_IF
        ELSE
            eBootStep := HOME_REF_OPT;
        END_IF
    HOME_REF_OPT:
        IF stChanParams.nReferencingOpt <> nRecentReferencingOpt THEN
            fbReferencingOptWrite.bExecute := TRUE;
            IF ftReferencingOptSetDone.Q THEN
                fbReferencingOptWrite.bExecute := FALSE;
                IF fbReferencingOptWrite.bError THEN
                    stMotionStage.bError   := fbReferencingOptWrite.bError;
                    stMotionStage.nErrorId := fbReferencingOptWrite.nErrId;
                    eBootStep              := ERR;
                ELSE
                    nRecentReferencingOpt := stChanParams.nReferencingOpt;
                    eBootStep             := STEPS;
                END_IF
            END_IF
        ELSE
            eBootStep := STEPS;
        END_IF

    // Step-mode params
    STEPS:
        IF nScalededSteps <> nRecentSteps THEN
            fbSetSteps.bExecute := TRUE;
            IF ftStepUpdateDone.Q THEN
                fbSetSteps.bExecute := FALSE;
                IF fbSetSteps.bError THEN
                    stMotionStage.bError   := fbSetSteps.bError;
                    stMotionStage.nErrorId := fbSetSteps.nErrId;
                    eBootStep              := ERR;
                ELSE
                    nRecentSteps := nScalededSteps;
                    eBootStep    := STEP_AMP;
                END_IF
            END_IF
        ELSE
            eBootStep := STEP_AMP;
        END_IF

    STEP_AMP:
        IF nScalededStepAmp <> nRecentStepAmp THEN
            fbSetStepAmp.bExecute := TRUE;
            IF ftStepAmpUpdateDone.Q THEN
                fbSetStepAmp.bExecute := FALSE;
                IF fbSetStepAmp.bError THEN
                    stMotionStage.bError   := fbSetStepAmp.bError;
                    stMotionStage.nErrorId := fbSetStepAmp.nErrId;
                    eBootStep              := ERR;
                ELSE
                    nRecentStepAmp := nScalededStepAmp;
                    eBootStep      := STEP_FREQ;
                END_IF
            END_IF
        ELSE
            eBootStep := STEP_FREQ;
        END_IF

    STEP_FREQ:
        IF nScaledStepFreq <> nRecentStepFreq THEN
            fbSetStepFreq.bExecute := TRUE;
            IF ftStepFreqUpdateDone.Q THEN
                fbSetStepFreq.bExecute := FALSE;
                IF fbSetStepFreq.bError THEN
                    stMotionStage.bError   := fbSetStepFreq.bError;
                    stMotionStage.nErrorId := fbSetStepFreq.nErrId;
                    eBootStep              := ERR;
                ELSE
                    nRecentStepFreq := nScaledStepFreq;
                    eBootStep       := DIST_CODE_INV;
                END_IF
            END_IF
        ELSE
            eBootStep := DIST_CODE_INV;
        END_IF

    // Extra channel params
    DIST_CODE_INV:
        IF stChanParams.nDistCodeInv <> nRecentDistCodeInv THEN
            fbDistCodeInvWrite.bExecute := TRUE;
            IF ftDistCodeInvSetDone.Q THEN
                fbDistCodeInvWrite.bExecute := FALSE;
                IF fbDistCodeInvWrite.bError THEN
                    stMotionStage.bError   := fbDistCodeInvWrite.bError;
                    stMotionStage.nErrorId := fbDistCodeInvWrite.nErrId;
                    eBootStep              := ERR;
                ELSE
                    nRecentDistCodeInv := stChanParams.nDistCodeInv;
                    eBootStep          := POS_CTRL_OPT;
                END_IF
            END_IF
        ELSE
            eBootStep := POS_CTRL_OPT;
        END_IF

    POS_CTRL_OPT:
        IF stChanParams.nPositionerCtrlOpt <> nRecentPositionerCtrlOpt THEN
            fbPositionerCtrlOptWrite.bExecute := TRUE;
            IF ftPositionerCtrlOptSetDone.Q THEN
                fbPositionerCtrlOptWrite.bExecute := FALSE;
                IF fbPositionerCtrlOptWrite.bError THEN
                    stMotionStage.bError   := fbPositionerCtrlOptWrite.bError;
                    stMotionStage.nErrorId := fbPositionerCtrlOptWrite.nErrId;
                    eBootStep              := ERR;
                ELSE
                    nRecentPositionerCtrlOpt := stChanParams.nPositionerCtrlOpt;
                    eBootStep                := ACT_MODE;
                END_IF
            END_IF
        ELSE
            eBootStep := ACT_MODE;
        END_IF

    ACT_MODE:
        IF stChanParams.nActuatorMode <> nRecentActuatorMode THEN
            fbActuatorModeWrite.bExecute := TRUE;
            IF ftActuatorModeSetDone.Q THEN
                fbActuatorModeWrite.bExecute := FALSE;
                IF fbActuatorModeWrite.bError THEN
                    stMotionStage.bError   := fbActuatorModeWrite.bError;
                    stMotionStage.nErrorId := fbActuatorModeWrite.nErrId;
                    eBootStep              := ERR;
                ELSE
                    nRecentActuatorMode := stChanParams.nActuatorMode;
                    eBootStep           := MOTOR_LOAD_PROT;
                END_IF
            END_IF
        ELSE
            eBootStep := MOTOR_LOAD_PROT;
        END_IF

    MOTOR_LOAD_PROT:
        IF stChanParams.nMotorLoadProt <> nRecentMotorLoadProt THEN
            fbMotorLoadProtWrite.bExecute := TRUE;
            IF ftMotorLoadProtSetDone.Q THEN
                fbMotorLoadProtWrite.bExecute := FALSE;
                IF fbMotorLoadProtWrite.bError THEN
                    stMotionStage.bError   := fbMotorLoadProtWrite.bError;
                    stMotionStage.nErrorId := fbMotorLoadProtWrite.nErrId;
                    eBootStep              := ERR;
                ELSE
                    nRecentMotorLoadProt := stChanParams.nMotorLoadProt;
                    eBootStep            := DONE;
                END_IF
            END_IF
        ELSE
            eBootStep := DONE;
        END_IF

    DONE:
        bBootSweepDone := TRUE;
        bSweepActive   := FALSE;
        bParamsSet     := TRUE;

    ERR:
        bSweepActive := FALSE;
        bParamsSet   := FALSE;

    ELSE
        eBootStep := IDLE;
END_CASE
END_METHOD

// Cyclic call of every SDO writer instance.
METHOD PRIVATE CallAllSdoWriters
// Channel
fbSetFErrorWin(
    sNetId     := stMotionStage.stAxisParameters.sAmsNetId,
    nSlaveAddr := stDS402Drive.nSlaveAddr,
    nIndex     := stChanParams.nChanFErrWinIdx,
    nSubIndex  := 0,
    pSrcBuf    := ADR(nScaledFErrWin),
    cbBufLen   := SIZEOF(nScaledFErrWin)
);
fbSetSoftLimMin(
    sNetId     := stMotionStage.stAxisParameters.sAmsNetId,
    nSlaveAddr := stDS402Drive.nSlaveAddr,
    nIndex     := stChanParams.nChanSoftLimitIdx,
    nSubIndex  := 1,
    pSrcBuf    := ADR(stChanParams.nSoftLimMin),
    cbBufLen   := SIZEOF(stChanParams.nSoftLimMin)
);
fbSetSoftLimMax(
    sNetId     := stMotionStage.stAxisParameters.sAmsNetId,
    nSlaveAddr := stDS402Drive.nSlaveAddr,
    nIndex     := stChanParams.nChanSoftLimitIdx,
    nSubIndex  := 2,
    pSrcBuf    := ADR(stChanParams.nSoftLimMax),
    cbBufLen   := SIZEOF(stChanParams.nSoftLimMax)
);
fbMaxCloseLoopFreqWrite(
    sNetId     := stMotionStage.stAxisParameters.sAmsNetId,
    nSlaveAddr := stDS402Drive.nSlaveAddr,
    nIndex     := stChanParams.nChanMaxCloseLoopFreqIdx,
    nSubIndex  := 0,
    pSrcBuf    := ADR(stChanParams.nMaxCloseLoopFreq),
    cbBufLen   := SIZEOF(stChanParams.nMaxCloseLoopFreq)
);
fbSensorPowerModeWrite(
    sNetId     := stMotionStage.stAxisParameters.sAmsNetId,
    nSlaveAddr := stDS402Drive.nSlaveAddr,
    nIndex     := stChanParams.nChanSensorPowerModeIdx,
    nSubIndex  := 0,
    pSrcBuf    := ADR(stChanParams.nSensorPowerMode),
    cbBufLen   := SIZEOF(stChanParams.nSensorPowerMode)
);
fbLogicalScaleOffsetWrite(
    sNetId     := stMotionStage.stAxisParameters.sAmsNetId,
    nSlaveAddr := stDS402Drive.nSlaveAddr,
    nIndex     := stChanParams.nChanLogicalScaleOfsIdx,
    nSubIndex  := 0,
    pSrcBuf    := ADR(stChanParams.nLogicalScaleOffset),
    cbBufLen   := SIZEOF(stChanParams.nLogicalScaleOffset)
);
fbLogicalScaleInvWrite(
    sNetId     := stMotionStage.stAxisParameters.sAmsNetId,
    nSlaveAddr := stDS402Drive.nSlaveAddr,
    nIndex     := stChanParams.nChanLogicalScaleInvIdx,
    nSubIndex  := 0,
    pSrcBuf    := ADR(stChanParams.nLogicalScaleInv),
    cbBufLen   := SIZEOF(stChanParams.nLogicalScaleInv)
);
fbSafeDirWrite(
    sNetId     := stMotionStage.stAxisParameters.sAmsNetId,
    nSlaveAddr := stDS402Drive.nSlaveAddr,
    nIndex     := stChanParams.nChanSafeDirIdx,
    nSubIndex  := 0,
    pSrcBuf    := ADR(stChanParams.nSafeDir),
    cbBufLen   := SIZEOF(stChanParams.nSafeDir)
);

// Calibration
fbCalibrationOptWrite(
    sNetId     := stMotionStage.stAxisParameters.sAmsNetId,
    nSlaveAddr := stDS402Drive.nSlaveAddr,
    nIndex     := stChanParams.nChanCalibrationOptIdx,
    nSubIndex  := 0,
    pSrcBuf    := ADR(stChanParams.nCalibrationOpt),
    cbBufLen   := SIZEOF(stChanParams.nCalibrationOpt)
);

// Home
fbSetHomeVeloFast(
    sNetId     := stMotionStage.stAxisParameters.sAmsNetId,
    nSlaveAddr := stDS402Drive.nSlaveAddr,
    nIndex     := stChanParams.nChanHomeVeloIdx,
    nSubIndex  := 1,
    pSrcBuf    := ADR(stChanParams.nHomeVeloFast),
    cbBufLen   := SIZEOF(stChanParams.nHomeVeloFast)
);
fbSetHomeVeloSlow(
    sNetId     := stMotionStage.stAxisParameters.sAmsNetId,
    nSlaveAddr := stDS402Drive.nSlaveAddr,
    nIndex     := stChanParams.nChanHomeVeloIdx,
    nSubIndex  := 2,
    pSrcBuf    := ADR(stChanParams.nHomeVeloSlow),
    cbBufLen   := SIZEOF(stChanParams.nHomeVeloSlow)
);
fbSetHomeAcc(
    sNetId     := stMotionStage.stAxisParameters.sAmsNetId,
    nSlaveAddr := stDS402Drive.nSlaveAddr,
    nIndex     := stChanParams.nChanhomeAccIdx,
    nSubIndex  := 0,
    pSrcBuf    := ADR(stChanParams.nHomeAcc),
    cbBufLen   := SIZEOF(stChanParams.nHomeAcc)
);
fbSetHomeOffs(
    sNetId     := stMotionStage.stAxisParameters.sAmsNetId,
    nSlaveAddr := stDS402Drive.nSlaveAddr,
    nIndex     := stChanParams.nChanHomeOffsIdx,
    nSubIndex  := 0,
    pSrcBuf    := ADR(stChanParams.nHomeOffset),
    cbBufLen   := SIZEOF(stChanParams.nHomeOffset)
);
fbSetHomeMethod(
    sNetId     := stMotionStage.stAxisParameters.sAmsNetId,
    nSlaveAddr := stDS402Drive.nSlaveAddr,
    nIndex     := stChanParams.nChanHomeMethodIdx,
    nSubIndex  := 0,
    pSrcBuf    := ADR(stChanParams.nHomeMethod),
    cbBufLen   := SIZEOF(stChanParams.nHomeMethod)
);
fbReferencingOptWrite(
    sNetId     := stMotionStage.stAxisParameters.sAmsNetId,
    nSlaveAddr := stDS402Drive.nSlaveAddr,
    nIndex     := stChanParams.nChanReferencingOptIdx,
    nSubIndex  := 0,
    pSrcBuf    := ADR(stChanParams.nReferencingOpt),
    cbBufLen   := SIZEOF(stChanParams.nReferencingOpt)
);

// Step-mode
fbSetSteps(
    sNetId     := stMotionStage.stAxisParameters.sAmsNetId,
    nSlaveAddr := stDS402Drive.nSlaveAddr,
    nIndex     := stChanParams.nChanStepIdx,
    nSubIndex  := 0,
    pSrcBuf    := ADR(nScalededSteps),
    cbBufLen   := SIZEOF(stChanParams.nChanStep)
);
fbSetStepAmp(
    sNetId     := stMotionStage.stAxisParameters.sAmsNetId,
    nSlaveAddr := stDS402Drive.nSlaveAddr,
    nIndex     := stChanParams.nChanStepAmpIdx,
    nSubIndex  := 0,
    pSrcBuf    := ADR(nScalededStepAmp),
    cbBufLen   := SIZEOF(stChanParams.nChanStepAmp)
);
fbSetStepFreq(
    sNetId     := stMotionStage.stAxisParameters.sAmsNetId,
    nSlaveAddr := stDS402Drive.nSlaveAddr,
    nIndex     := stChanParams.nChanStepFreqIdx,
    nSubIndex  := 0,
    pSrcBuf    := ADR(nScaledStepFreq),
    cbBufLen   := SIZEOF(stChanParams.nChanStepFreq)
);

// Extra channel params
fbDistCodeInvWrite(
    sNetId     := stMotionStage.stAxisParameters.sAmsNetId,
    nSlaveAddr := stDS402Drive.nSlaveAddr,
    nIndex     := stChanParams.nChanDistCodeInvIdx,
    nSubIndex  := 0,
    pSrcBuf    := ADR(stChanParams.nDistCodeInv),
    cbBufLen   := SIZEOF(stChanParams.nDistCodeInv)
);
fbPositionerCtrlOptWrite(
    sNetId     := stMotionStage.stAxisParameters.sAmsNetId,
    nSlaveAddr := stDS402Drive.nSlaveAddr,
    nIndex     := stChanParams.nChanPositionerCtrlOptIdx,
    nSubIndex  := 0,
    pSrcBuf    := ADR(stChanParams.nPositionerCtrlOpt),
    cbBufLen   := SIZEOF(stChanParams.nPositionerCtrlOpt)
);
fbActuatorModeWrite(
    sNetId     := stMotionStage.stAxisParameters.sAmsNetId,
    nSlaveAddr := stDS402Drive.nSlaveAddr,
    nIndex     := stChanParams.nChanActuatorModeIdx,
    nSubIndex  := 0,
    pSrcBuf    := ADR(stChanParams.nActuatorMode),
    cbBufLen   := SIZEOF(stChanParams.nActuatorMode)
);
fbMotorLoadProtWrite(
    sNetId     := stMotionStage.stAxisParameters.sAmsNetId,
    nSlaveAddr := stDS402Drive.nSlaveAddr,
    nIndex     := stChanParams.nChanMotorLoadProtIdx,
    nSubIndex  := 0,
    pSrcBuf    := ADR(stChanParams.nMotorLoadProt),
    cbBufLen   := SIZEOF(stChanParams.nMotorLoadProt)
);
END_METHOD

// Pre-boot / fault state: clear every bExecute so no SDO writes go out.
// CallAllSdoWriters still ticks each FB cyclically (required by Beckhoff
// CoE writer semantics), but with bExecute=FALSE they remain idle.
METHOD PRIVATE HoldAllWritersIdle
fbSetFErrorWin.bExecute            := FALSE;
fbSetSoftLimMin.bExecute           := FALSE;
fbSetSoftLimMax.bExecute           := FALSE;
fbMaxCloseLoopFreqWrite.bExecute   := FALSE;
fbSensorPowerModeWrite.bExecute    := FALSE;
fbLogicalScaleOffsetWrite.bExecute := FALSE;
fbLogicalScaleInvWrite.bExecute    := FALSE;
fbSafeDirWrite.bExecute            := FALSE;
fbCalibrationOptWrite.bExecute     := FALSE;
fbSetHomeVeloFast.bExecute         := FALSE;
fbSetHomeVeloSlow.bExecute         := FALSE;
fbSetHomeAcc.bExecute              := FALSE;
fbSetHomeOffs.bExecute             := FALSE;
fbSetHomeMethod.bExecute           := FALSE;
fbReferencingOptWrite.bExecute     := FALSE;
fbSetSteps.bExecute                := FALSE;
fbSetStepAmp.bExecute              := FALSE;
fbSetStepFreq.bExecute             := FALSE;
fbDistCodeInvWrite.bExecute        := FALSE;
fbPositionerCtrlOptWrite.bExecute  := FALSE;
fbActuatorModeWrite.bExecute       := FALSE;
fbMotorLoadProtWrite.bExecute      := FALSE;
END_METHOD

// Runtime: monitor every parameter; when the setpoint diverges from the
// cached value, fire its SDO write. Independent per parameter.
METHOD PRIVATE ParallelOnDemand
CASE stChanParams.eHomeMode OF
E_MCS2HomeMethod.AutoMethod:
    stChanParams.nLogicalScaleOffset := DINT_TO_UDINT(stChanParams.nHomeOffset);
END_CASE

fbSetFErrorWin.bExecute            := nScaledFErrWin                   <> nRecentFErrWin;
fbSetSoftLimMin.bExecute           := stChanParams.nSoftLimMin         <> nRecentSoftLimMin;
fbSetSoftLimMax.bExecute           := stChanParams.nSoftLimMax         <> nRecentSoftLimMax;
fbMaxCloseLoopFreqWrite.bExecute   := stChanParams.nMaxCloseLoopFreq   <> nRecentMaxCloseLoopFreq;
fbSensorPowerModeWrite.bExecute    := stChanParams.nSensorPowerMode    <> nRecentSensorPowerMode;
fbLogicalScaleOffsetWrite.bExecute := stChanParams.nLogicalScaleOffset <> nRecentLogicalScaleOffset;
fbLogicalScaleInvWrite.bExecute    := bInPreOp AND (stChanParams.nLogicalScaleInv <> nRecentLogicalScaleInv);
fbSafeDirWrite.bExecute            := bInPreOp AND (stChanParams.nSafeDir <> nRecentSafeDir);
fbCalibrationOptWrite.bExecute     := stChanParams.nCalibrationOpt     <> nRecentCalibrationOpt;
fbSetHomeVeloFast.bExecute         := stChanParams.nHomeVeloFast       <> nRecentHomeVeloFast;
fbSetHomeVeloSlow.bExecute         := stChanParams.nHomeVeloSlow       <> nRecentHomeVeloSlow;
fbSetHomeAcc.bExecute              := stChanParams.nHomeAcc            <> nRecentHomeAcc;
fbSetHomeOffs.bExecute             := stChanParams.nHomeOffset         <> nRecentHomeOffset;
fbSetHomeMethod.bExecute           := stChanParams.nHomeMethod         <> nRecentHomeMethod;
fbReferencingOptWrite.bExecute     := stChanParams.nReferencingOpt     <> nRecentReferencingOpt;
fbSetSteps.bExecute                := nScalededSteps				   <> nRecentSteps;
fbSetStepAmp.bExecute              := nScalededStepAmp                 <> nRecentStepAmp;
fbSetStepFreq.bExecute             := nScaledStepFreq                  <> nRecentStepFreq;
fbDistCodeInvWrite.bExecute        := stChanParams.nDistCodeInv        <> nRecentDistCodeInv;
fbPositionerCtrlOptWrite.bExecute  := stChanParams.nPositionerCtrlOpt  <> nRecentPositionerCtrlOpt;
fbActuatorModeWrite.bExecute       := stChanParams.nActuatorMode       <> nRecentActuatorMode;
fbMotorLoadProtWrite.bExecute      := stChanParams.nMotorLoadProt      <> nRecentMotorLoadProt;

// On any completion edge, latch the new cached value and clear errors.
IF ftFErrWinSetDone.Q THEN
    IF fbSetFErrorWin.bError THEN
        stMotionStage.bError   := fbSetFErrorWin.bError;
        stMotionStage.nErrorId := fbSetFErrorWin.nErrId;
    ELSE
        nRecentFErrWin := nScaledFErrWin;
    END_IF
    fbSetFErrorWin.bExecute := FALSE;
END_IF
IF ftSoftLimMinSetDone.Q THEN
    IF fbSetSoftLimMin.bError THEN
        stMotionStage.bError   := fbSetSoftLimMin.bError;
        stMotionStage.nErrorId := fbSetSoftLimMin.nErrId;
    ELSE
        nRecentSoftLimMin := stChanParams.nSoftLimMin;
    END_IF
    fbSetSoftLimMin.bExecute := FALSE;
END_IF
IF ftSoftLimMaxSetDone.Q THEN
    IF fbSetSoftLimMax.bError THEN
        stMotionStage.bError   := fbSetSoftLimMax.bError;
        stMotionStage.nErrorId := fbSetSoftLimMax.nErrId;
    ELSE
        nRecentSoftLimMax := stChanParams.nSoftLimMax;
    END_IF
    fbSetSoftLimMax.bExecute := FALSE;
END_IF
IF ftMaxCloseLoopFreqSetDone.Q THEN
    IF fbMaxCloseLoopFreqWrite.bError THEN
        stMotionStage.bError   := fbMaxCloseLoopFreqWrite.bError;
        stMotionStage.nErrorId := fbMaxCloseLoopFreqWrite.nErrId;
    ELSE
        nRecentMaxCloseLoopFreq := stChanParams.nMaxCloseLoopFreq;
    END_IF
    fbMaxCloseLoopFreqWrite.bExecute := FALSE;
END_IF
IF ftSensorPowerModeSetDone.Q THEN
    IF fbSensorPowerModeWrite.bError THEN
        stMotionStage.bError   := fbSensorPowerModeWrite.bError;
        stMotionStage.nErrorId := fbSensorPowerModeWrite.nErrId;
    ELSE
        nRecentSensorPowerMode := stChanParams.nSensorPowerMode;
    END_IF
    fbSensorPowerModeWrite.bExecute := FALSE;
END_IF
IF ftLogicalScaleOffsetSetDone.Q THEN
    IF fbLogicalScaleOffsetWrite.bError THEN
        stMotionStage.bError   := fbLogicalScaleOffsetWrite.bError;
        stMotionStage.nErrorId := fbLogicalScaleOffsetWrite.nErrId;
    ELSE
        nRecentLogicalScaleOffset := stChanParams.nLogicalScaleOffset;
    END_IF
    fbLogicalScaleOffsetWrite.bExecute := FALSE;
END_IF
IF ftLogicalScaleInvSetDone.Q THEN
    IF fbLogicalScaleInvWrite.bError THEN
        stMotionStage.bError   := fbLogicalScaleInvWrite.bError;
        stMotionStage.nErrorId := fbLogicalScaleInvWrite.nErrId;
    ELSE
        nRecentLogicalScaleInv := stChanParams.nLogicalScaleInv;
    END_IF
    fbLogicalScaleInvWrite.bExecute := FALSE;
END_IF
IF ftSafeDirSetDone.Q THEN
    IF fbSafeDirWrite.bError THEN
        stMotionStage.bError   := fbSafeDirWrite.bError;
        stMotionStage.nErrorId := fbSafeDirWrite.nErrId;
    ELSE
        nRecentSafeDir := stChanParams.nSafeDir;
    END_IF
    fbSafeDirWrite.bExecute := FALSE;
END_IF
IF ftCalibrationOptSetDone.Q THEN
    IF fbCalibrationOptWrite.bError THEN
        stMotionStage.bError   := fbCalibrationOptWrite.bError;
        stMotionStage.nErrorId := fbCalibrationOptWrite.nErrId;
    ELSE
        nRecentCalibrationOpt := stChanParams.nCalibrationOpt;
    END_IF
    fbCalibrationOptWrite.bExecute := FALSE;
END_IF
IF ftHomeVeloFastSetDone.Q THEN
    IF fbSetHomeVeloFast.bError THEN
        stMotionStage.bError   := fbSetHomeVeloFast.bError;
        stMotionStage.nErrorId := fbSetHomeVeloFast.nErrId;
    ELSE
        nRecentHomeVeloFast := stChanParams.nHomeVeloFast;
    END_IF
    fbSetHomeVeloFast.bExecute := FALSE;
END_IF
IF ftHomeVeloSlowSetDone.Q THEN
    IF fbSetHomeVeloSlow.bError THEN
        stMotionStage.bError   := fbSetHomeVeloSlow.bError;
        stMotionStage.nErrorId := fbSetHomeVeloSlow.nErrId;
    ELSE
        nRecentHomeVeloSlow := stChanParams.nHomeVeloSlow;
    END_IF
    fbSetHomeVeloSlow.bExecute := FALSE;
END_IF
IF ftHomeAccSetDone.Q THEN
    IF fbSetHomeAcc.bError THEN
        stMotionStage.bError   := fbSetHomeAcc.bError;
        stMotionStage.nErrorId := fbSetHomeAcc.nErrId;
    ELSE
        nRecentHomeAcc := stChanParams.nHomeAcc;
    END_IF
    fbSetHomeAcc.bExecute := FALSE;
END_IF
IF ftHomeOffsSetDone.Q THEN
    IF fbSetHomeOffs.bError THEN
        stMotionStage.bError   := fbSetHomeOffs.bError;
        stMotionStage.nErrorId := fbSetHomeOffs.nErrId;
    ELSE
        nRecentHomeOffset := stChanParams.nHomeOffset;
    END_IF
    fbSetHomeOffs.bExecute := FALSE;
END_IF
IF ftReferencingOptSetDone.Q THEN
    IF fbReferencingOptWrite.bError THEN
        stMotionStage.bError   := fbReferencingOptWrite.bError;
        stMotionStage.nErrorId := fbReferencingOptWrite.nErrId;
    ELSE
        nRecentReferencingOpt := stChanParams.nReferencingOpt;
    END_IF
    fbReferencingOptWrite.bExecute := FALSE;
END_IF
IF ftStepUpdateDone.Q THEN
    IF fbSetSteps.bError THEN
        stMotionStage.bError   := fbSetSteps.bError;
        stMotionStage.nErrorId := fbSetSteps.nErrId;
    ELSE
        nRecentSteps := nScalededSteps;
    END_IF
    fbSetSteps.bExecute := FALSE;
END_IF
IF ftStepAmpUpdateDone.Q THEN
    IF fbSetStepAmp.bError THEN
        stMotionStage.bError   := fbSetStepAmp.bError;
        stMotionStage.nErrorId := fbSetStepAmp.nErrId;
    ELSE
        nRecentStepAmp := nScalededStepAmp;
    END_IF
    fbSetStepAmp.bExecute := FALSE;
END_IF
IF ftStepFreqUpdateDone.Q THEN
    IF fbSetStepFreq.bError THEN
        stMotionStage.bError   := fbSetStepFreq.bError;
        stMotionStage.nErrorId := fbSetStepFreq.nErrId;
    ELSE
        nRecentStepFreq := nScaledStepFreq;
    END_IF
    fbSetStepFreq.bExecute := FALSE;
END_IF
IF ftDistCodeInvSetDone.Q THEN
    IF fbDistCodeInvWrite.bError THEN
        stMotionStage.bError   := fbDistCodeInvWrite.bError;
        stMotionStage.nErrorId := fbDistCodeInvWrite.nErrId;
    ELSE
        nRecentDistCodeInv := stChanParams.nDistCodeInv;
    END_IF
    fbDistCodeInvWrite.bExecute := FALSE;
END_IF
IF ftPositionerCtrlOptSetDone.Q THEN
    IF fbPositionerCtrlOptWrite.bError THEN
        stMotionStage.bError   := fbPositionerCtrlOptWrite.bError;
        stMotionStage.nErrorId := fbPositionerCtrlOptWrite.nErrId;
    ELSE
        nRecentPositionerCtrlOpt := stChanParams.nPositionerCtrlOpt;
    END_IF
    fbPositionerCtrlOptWrite.bExecute := FALSE;
END_IF
IF ftActuatorModeSetDone.Q THEN
    IF fbActuatorModeWrite.bError THEN
        stMotionStage.bError   := fbActuatorModeWrite.bError;
        stMotionStage.nErrorId := fbActuatorModeWrite.nErrId;
    ELSE
        nRecentActuatorMode := stChanParams.nActuatorMode;
    END_IF
    fbActuatorModeWrite.bExecute := FALSE;
END_IF
IF ftMotorLoadProtSetDone.Q THEN
    IF fbMotorLoadProtWrite.bError THEN
        stMotionStage.bError   := fbMotorLoadProtWrite.bError;
        stMotionStage.nErrorId := fbMotorLoadProtWrite.nErrId;
    ELSE
        nRecentMotorLoadProt := stChanParams.nMotorLoadProt;
    END_IF
    fbMotorLoadProtWrite.bExecute := FALSE;
END_IF
END_METHOD

METHOD PRIVATE ScaleDriveParams
nScaledFErrWin := LREAL_TO_DINT(
    stMotionStage.stAxisParameters.fCtrlPosDiffMax
    / MAX(stMotionStage.stAxisParameters.fEncScaleFactorInternal,
          stChanParams.fScalingFactor));

IF stMotionStage.stAxisParameters.bEncEnableSoftEndMinControl.0
   AND stMotionStage.stAxisParameters.bEncEnableSoftEndMaxControl.0 THEN
    stChanParams.nSoftLimMax := LREAL_TO_DINT(
        stMotionStage.stAxisParameters.fEncSoftEndMax
        / MAX(stMotionStage.stAxisParameters.fEncScaleFactorInternal,
              stChanParams.fScalingFactor));
    stChanParams.nSoftLimMin := LREAL_TO_DINT(
        stMotionStage.stAxisParameters.fEncSoftEndMin
        / MAX(stMotionStage.stAxisParameters.fEncScaleFactorInternal,
              stChanParams.fScalingFactor));
ELSE
    stChanParams.nSoftLimMax := 0;
    stChanParams.nSoftLimMin := 0;
END_IF
END_METHOD

METHOD PRIVATE ScaleHomingParams
CASE stChanParams.eHomeMode OF
    E_MCS2HomeMethod.AutoMethod,E_MCS2HomeMethod.CurrentPositionMethod:
        stChanParams.nHomeVeloFast := LREAL_TO_UDINT(
            stMotionStage.stAxisParameters.fRefVeloSearch
            / MAX(stMotionStage.stAxisParameters.fEncScaleFactorInternal,
                  stChanParams.fScalingFactor));

        stChanParams.nHomeVeloSlow := LREAL_TO_UDINT(
            stMotionStage.stAxisParameters.fRefVeloSync
            / MAX(stMotionStage.stAxisParameters.fEncScaleFactorInternal,
                  stChanParams.fScalingFactor));

        stChanParams.nHomeAcc := LREAL_TO_UDINT(
            stChanParams.fHomeAcc
            / MAX(stMotionStage.stAxisParameters.fEncScaleFactorInternal,
                  stChanParams.fScalingFactor));

        stChanParams.nHomeOffset := LREAL_TO_DINT(
            stMotionStage.fHomePosition
            / MAX(stMotionStage.stAxisParameters.fEncScaleFactorInternal,
                  stChanParams.fScalingFactor));

        stChanParams.nHomeMethod := TO_SINT(stChanParams.eHomeMode);

END_CASE
END_METHOD

METHOD PRIVATE ScaleStepModeParams
nScalededSteps   := LIMIT(-1000, stChanParams.nChanStep, 1000);
nScalededStepAmp := REAL_TO_UINT(LIMIT(50,  stChanParams.nChanStepAmp,  100) * 655.35);
nScaledStepFreq  := REAL_TO_UINT(LIMIT(500, stChanParams.nChanStepFreq, 1000.0));
END_METHOD

END_FUNCTION_BLOCK

// ---- POUs/Motion/DS402/MCS2/FB_ReadDriveCodes.TcPOU
(* Read Drive error codes after a motion or fault condition occured *)
FUNCTION_BLOCK FB_ReadDriveCodes
VAR_IN_OUT
    stDS402Drive         : ST_DS402Drive;
    stMotionStage        : ST_MotionStage;
    stMCS2ChanParameter	: ST_MCS2ChanParameter;
END_VAR
VAR_INPUT
    bEnable : BOOL;
END_VAR
VAR
    {attribute 'hide'}
    fbLogError          : FB_LogMotionError;
    sMsg                : STRING;
    sMCS2Code           : STRING;
    bMCS2Fault          : BOOL;
    rtMCS2Fault         : R_TRIG;
END_VAR

IF NOT __ISVALIDREF(stDS402Drive)
    OR NOT __ISVALIDREF(stMotionStage)
    OR NOT __ISVALIDREF(stMCS2ChanParameter) THEN
    RETURN;
END_IF

// The drive-side code (0x603F) is read by FB_ReadChanParameters on a fault or
// internal-limit event. It is decoded by its own table and never merged into
// nErrorId: the two number spaces overlap (MCS2 0x4200 sits inside the NC 0x4xxx
// family, and MCS2 manufacturer codes 0xFFxx overlap E_LCLSMotionError.TEST).
// The decoded string and raw code stay on MCS2_ERR_MSG / MCS2_ERR for PLC debug;
// only the raw code is surfaced to the operator via sErrorMessage below.
stMCS2ChanParameter.sMCS2ErrorMessage :=
    F_MCS2ErrorCodeLookup(nErrorId := stMCS2ChanParameter.nMCS2ErrorCode);

// Promote a genuine MCS2 fault the NC never latched (a drive-side stop that
// does not disturb the NC position loop). Only real-time conditions qualify,
// checked in any op mode: Overload/OverTemperature/PositionerFault hold for as
// long as the condition is physically present, and FollowingLimitReached is
// the firmware's own Following Error Window (0x6065) protective stop, which
// it enforces continuously, including during CSP streaming.
//
// MovementFailed is excluded: it describes the outcome of a discrete
// MCS2-native move (home/step/calibrate), which CSP never issues. CSP only
// streams continuous setpoints, so in CSP that bit can only ever be a stale
// leftover from an earlier open-loop move, not a live result, and surfacing
// it there faulted CSP moves that had actually succeeded. The open-loop
// routines already detect their own move failures via the DS402 status word
// (see FB_MCS2Home/FB_MCS2StepMode/FB_MCS2Calibrate).
//
// Edge-triggered so it reports once: a reset clears bError, and a
// still-asserted condition does not re-latch and block the reset. A fresh
// fault re-fires on the next rising edge.
bMCS2Fault :=
    bEnable
    AND (stMCS2ChanParameter.stChannelState.bFollowingLimitReached
         OR stMCS2ChanParameter.stChannelState.bPositionerOverload
         OR stMCS2ChanParameter.stChannelState.bOverTemperature
         OR stMCS2ChanParameter.stChannelState.bPositionerFault);

rtMCS2Fault(CLK := bMCS2Fault);
IF rtMCS2Fault.Q AND NOT stMotionStage.bError THEN
    stMotionStage.bError   S= TRUE;
    stMotionStage.nErrorId := E_LCLSMotionError.MCS2_FAULT;
END_IF

// sErrorMessage is the only message channel exposed to the IOC. Rebuild it from
// scratch each cycle so the MCS2 layer, an SDO read that lands several cycles
// after bError latches, merges in exactly once it is available, without ever
// duplicating. The numeric values stay separate in PLC:nErrorId and MCS2_ERR so
// the overlapping code spaces cannot be confused.
IF stMotionStage.bError THEN
    sMsg := '';

    // NC / limit layer: whatever the NC side could see.
    IF stDS402Drive.stDriveStatus.InternalLimitActive
        AND stMotionStage.sCustomErrorMessage <> '' THEN
        sMsg := stMotionStage.sCustomErrorMessage;
    ELSIF stMotionStage.nErrorId >= 16#4000 THEN
        sMsg := F_MotionErrorCodeLookup(nErrorId := stMotionStage.nErrorId);
    ELSIF stMotionStage.sCustomErrorMessage <> '' THEN
        sMsg := stMotionStage.sCustomErrorMessage;
    ELSIF stMotionStage.nErrorId = 0 AND stMCS2ChanParameter.nMCS2ErrorCode = 0 THEN
        sMsg := 'Contact PCDS to add new message';
    END_IF

    // MCS2 layer: append the raw drive code (hex) whenever one exists.
    IF stMCS2ChanParameter.nMCS2ErrorCode <> 0 THEN
        sMCS2Code := CONCAT('MCS2: 0x',
            WORD_TO_HEXSTR(in := stMCS2ChanParameter.nMCS2ErrorCode, iPrecision := 4, bLoCase := 0));
        IF sMsg <> '' THEN
            sMsg := CONCAT(CONCAT(sMsg, ' ('), CONCAT(sMCS2Code, ')'));
        ELSE
            sMsg := sMCS2Code;
        END_IF
    END_IF

    IF sMsg <> '' THEN
        stMotionStage.sErrorMessage := sMsg;
    END_IF
END_IF

END_FUNCTION_BLOCK

// ---- POUs/Motion/DS402/MCS2/F_MCS2ErrorCodeLookup.TcPOU
(*
    Decode an MCS2 drive error code read from the Error Code object (0x603F).
    Separate from F_MotionErrorCodeLookup on purpose: MCS2/DS402 codes and TwinCAT
    NC codes occupy overlapping numeric ranges (MCS2 0x4200 sits inside the NC
    0x4xxx family), so the two tables must never be applied to the same value.
    Codes per MCS2 EtherCAT Interface User Manual, appendix A.1.
*)
FUNCTION F_MCS2ErrorCodeLookup : STRING
VAR_INPUT
    nErrorId : UINT;
END_VAR
VAR
    msg : STRING;
    nClass : BYTE;
END_VAR

CASE nErrorId OF
    // DS402-mapped errors
    16#0000: msg := '';
    16#1000: msg := 'General error (unspecified MCS2 error)';
    16#1080: msg := 'Not ready for operation: amplifier disabled';
    16#3230: msg := 'Load error: positioner overload';
    16#4200: msg := 'Temperature error: over temperature';
    16#5100: msg := 'Supply error: power supply disabled';
    16#6100: msg := 'Internal software error';
    16#6320: msg := 'Parameter error: invalid parameter';
    16#7100: msg := 'Power error: supply failure or overload';
    16#7121: msg := 'Motor blocked: end stop reached';
    16#7300: msg := 'Sensor error: missing, disabled or unsupported type';
    16#7320: msg := 'Sensor position: no sensor present';
    16#7500: msg := 'Internal communication fault';
    16#8311: msg := 'Excess torque: control loop unstable';
    16#8500: msg := 'Range limit reached';
    // Not in manual table A.1, but what the drive reports over EtherCAT once a
    // move is aborted. It names the failed move, not the cause: read the channel
    // state RANGE_LIMIT / END_STOP bits to tell a soft limit from an end stop.
    16#8600: msg := 'Movement failed';
    16#8611: msg := 'Following error limit reached';

    // Manufacturer specific errors
    16#FF00: msg := 'Timeout';
    16#FF01: msg := 'Invalid data';
    16#FF02: msg := 'Aborted';
    16#FF03: msg := 'Permission denied';
    16#FF04: msg := 'Movement locked';
    16#FF05: msg := 'Overrange';
    16#FF06: msg := 'Invalid configuration';
    16#FF07: msg := 'Invalid sensor mode';
    16#FF08: msg := 'Invalid actuator mode';
    16#FF09: msg := 'Invalid control options';
    16#FF21: msg := 'Internal communication';

    ELSE
        // Table A.1 is not exhaustive, so fall back to the DS402 error class in
        // the high byte rather than reporting nothing useful.
        nClass := UINT_TO_BYTE(SHR(nErrorId, 8));
        CASE nClass OF
            16#10:                      msg := 'Generic error';
            16#20, 16#21, 16#22, 16#23: msg := 'Current error';
            16#30, 16#31, 16#32, 16#33: msg := 'Voltage error';
            16#40, 16#41, 16#42:        msg := 'Temperature error';
            16#50:                      msg := 'Device hardware error';
            16#60, 16#61, 16#62, 16#63: msg := 'Device software error';
            16#70:                      msg := 'Additional modules error';
            16#80:                      msg := 'Monitoring error';
            16#81:                      msg := 'Communication error';
            16#82:                      msg := 'Protocol error';
            16#83:                      msg := 'Torque control error';
            16#84:                      msg := 'Velocity controller error';
            16#85:                      msg := 'Position controller error';
            16#86:                      msg := 'Movement failed';
            16#87:                      msg := 'Sync controller error';
            16#90:                      msg := 'External error';
            16#F0:                      msg := 'Additional functions error';
            16#FF:                      msg := CONCAT('Device specific error (0x',
                            CONCAT(WORD_TO_HEXSTR(in := nErrorId, iPrecision := 4, bLoCase := 0),
                              ')'));
            ELSE
                msg := 'Unknown MCS2 error code';
        END_CASE
END_CASE

F_MCS2ErrorCodeLookup := msg;

END_FUNCTION

// ---- POUs/Motion/DS402/MCS2/FB_WriteCalibrationParameters.TcPOU
// Calibration Param SDO Hybrid Logic (startup-sequential, then on-demand)
// Sequential trigger (bCalibParamStep statemachine) is used at startup or force, otherwise parallel/on-demand.

FUNCTION_BLOCK FB_WriteCalibrationParameters
VAR_INPUT
    bEnable : BOOL;
END_VAR
VAR_IN_OUT
    stDS402Drive         : ST_DS402Drive;
    stMotionStage        : ST_MotionStage;
    stMCS2ChanParameter	: ST_MCS2ChanParameter;
END_VAR

VAR_OUTPUT
   bCalibrationsParamsSet : BOOL;
END_VAR
VAR
    {attribute 'hide'}
    fbChannelTypeWrite          : FB_EcCoESdoWrite;
    {attribute 'hide'}
    fbPositionerTypeWrite       : FB_EcCoESdoWrite;
    {attribute 'hide'}
    fbCalibrationOptWrite       : FB_EcCoESdoWrite;
    {attribute 'hide'}
    ftPositionerTypeSetDone     : F_TRIG;
    {attribute 'hide'}
    ftCalibrationOptSetDone     : F_TRIG;
    {attribute 'hide'}
    ftChannelTypeSetDone        : F_TRIG;
    {attribute 'hide'}
    nRecentPositionerType       : UDINT;
    {attribute 'hide'}
    nRecentCalibrationOpt       : UDINT;
    {attribute 'hide'}
    nRecentChannelType          : UDINT;
    tonStartUp : TON;
    nCalibParamStep : (IDLE := 0, CALIBOPTS := 1, DONE := 10, ERROR := -1) := IDLE;
    bForceSequentialSDOs : BOOL := FALSE;
    bErrorAcknowledge: BOOL;
END_VAR

IF NOT __ISVALIDREF(stDS402Drive)
    OR NOT __ISVALIDREF(stMotionStage)
    OR NOT __ISVALIDREF(stMCS2ChanParameter) THEN
    RETURN;
END_IF

IF bEnable THEN
    tonStartUp(
        IN := bEnable AND NOT bCalibrationsParamsSet,
        PT := T#6S
    );

    // Reset sequence if startup timer hasn't fired and not forcing sequential SDOs
    IF NOT tonStartUp.Q AND nCalibParamStep <> IDLE AND NOT bForceSequentialSDOs THEN
        nCalibParamStep := IDLE;
    END_IF

    // Acknowledge error and restart sequence
    IF nCalibParamStep = ERROR AND bErrorAcknowledge THEN
        nCalibParamStep        := IDLE;
        stMotionStage.bError   := FALSE;
        stMotionStage.nErrorId := 0;
    END_IF

    ftCalibrationOptSetDone(CLK := fbCalibrationOptWrite.bBusy);

    IF tonStartUp.Q OR bForceSequentialSDOs THEN
        CASE nCalibParamStep OF
            IDLE:
                bCalibrationsParamsSet         := FALSE;
                fbCalibrationOptWrite.bExecute := FALSE;
                nCalibParamStep                := CALIBOPTS;

            CALIBOPTS: // Calibration Option
                IF stMCS2ChanParameter.nCalibrationOpt <> nRecentCalibrationOpt THEN
                    fbCalibrationOptWrite.bExecute := TRUE;
                    IF ftCalibrationOptSetDone.Q THEN
                        fbCalibrationOptWrite.bExecute := FALSE;
                        IF fbCalibrationOptWrite.bError THEN
                            stMotionStage.bError   := fbCalibrationOptWrite.bError;
                            stMotionStage.nErrorId := fbCalibrationOptWrite.nErrId;
                            nCalibParamStep        := ERROR;
                        ELSE
                            nRecentCalibrationOpt := stMCS2ChanParameter.nCalibrationOpt;
                            nCalibParamStep       := DONE;
                        END_IF
                    END_IF
                ELSE
                    nCalibParamStep := DONE;
                END_IF

            DONE:
                bCalibrationsParamsSet := TRUE;

            ERROR:
                bCalibrationsParamsSet := FALSE;

            ELSE
                nCalibParamStep := IDLE;
        END_CASE

    ELSE
        // Parallel SDO mode — single write
        fbCalibrationOptWrite.bExecute := stMCS2ChanParameter.nCalibrationOpt <> nRecentCalibrationOpt;
        IF ftCalibrationOptSetDone.Q THEN
            fbCalibrationOptWrite.bExecute := FALSE;
            IF fbCalibrationOptWrite.bError THEN
                stMotionStage.bError   := fbCalibrationOptWrite.bError;
                stMotionStage.nErrorId := fbCalibrationOptWrite.nErrId;
            ELSE
                nRecentCalibrationOpt  := stMCS2ChanParameter.nCalibrationOpt;
                bCalibrationsParamsSet := TRUE;
            END_IF
        END_IF
    END_IF

    fbCalibrationOptWrite(
        sNetId     := stMotionStage.stAxisParameters.sAmsNetId,
        nSlaveAddr := stDS402Drive.nSlaveAddr,
        nIndex     := stMCS2ChanParameter.nChanCalibrationOptIdx,
        nSubIndex  := 0,
        pSrcBuf    := ADR(stMCS2ChanParameter.nCalibrationOpt),
        cbBufLen   := SIZEOF(stMCS2ChanParameter.nCalibrationOpt)
    );

    bCalibrationsParamsSet R= fbCalibrationOptWrite.bBusy;
END_IF

END_FUNCTION_BLOCK

// ---- POUs/Motion/DS402/MCS2/FB_WriteHomeParameters.TcPOU
// The SDO writes can be done sequentially at boot or on demand during normal use.
// Set bForceSequentialSDOs TRUE (debug) to enforce sequential behavior at any time.
FUNCTION_BLOCK FB_WriteHomeParameters
VAR_INPUT
    bEnable : BOOL;
END_VAR
VAR_IN_OUT
    stDS402Drive         : ST_DS402Drive;
    stMotionStage        : ST_MotionStage;
    stMCS2ChanParameter	: ST_MCS2ChanParameter;
END_VAR

VAR_OUTPUT
   bHomingParamsSet : BOOL;
END_VAR
VAR
    nHomingStep : (IDLE := 0, VELO_FAST := 1, VELO_SLOW := 2, ACC := 3, OFFSET := 4, REF_OPT := 5, DONE := 10, ERROR := -1) := IDLE;
    bForceSequentialSDOs : BOOL := FALSE;
    {attribute 'hide'}
    fbSetHomeOffs               : FB_EcCoESdoWrite;
    {attribute 'hide'}
    fbSetHomeVeloFast           : FB_EcCoESdoWrite;
    {attribute 'hide'}
    fbSetHomeVeloSlow           : FB_EcCoESdoWrite;
    {attribute 'hide'}
    fbSetHomeAcc                : FB_EcCoESdoWrite;
    {attribute 'hide'}
    fbReferencingOptWrite       : FB_EcCoESdoWrite;
    {attribute 'hide'}
    ftHomeVeloFastSetDone       : F_TRIG;
    {attribute 'hide'}
    ftHomeAccSetDone            : F_TRIG;
    {attribute 'hide'}
    ftHomeOffsSetDone           : F_TRIG;
    {attribute 'hide'}
    ftHomeVeloSlowSetDone       : F_TRIG;
    {attribute 'hide'}
    ftReferencingOptSetDone     : F_TRIG;

    {attribute 'hide'}
    nRecentHomeVeloFast         : UDINT;
    {attribute 'hide'}
    nRecentHomeVeloSlow         : UDINT;
    {attribute 'hide'}
    nRecentHomeAcc              : UDINT;
    {attribute 'hide'}
    nRecentHomeOffset           : DINT;
    {attribute 'hide'}
    nRecentReferencingOpt       : UDINT;
    {attribute 'hide'}
    nHomeOffs                   : DINT;
    tonStartUp : TON;
    bErrorAcknowledge: BOOL;
END_VAR

IF NOT __ISVALIDREF(stDS402Drive)
    OR NOT __ISVALIDREF(stMotionStage)
    OR NOT __ISVALIDREF(stMCS2ChanParameter) THEN
    RETURN;
END_IF

IF bEnable THEN
    tonStartUp(
        IN := bEnable AND NOT bHomingParamsSet,
        PT := T#4S
    );

    IF NOT tonStartUp.Q AND nHomingStep <> IDLE AND NOT bForceSequentialSDOs THEN
        nHomingStep := IDLE;
    END_IF

    IF nHomingStep = ERROR AND bErrorAcknowledge THEN
        nHomingStep            := IDLE;
        stMotionStage.bError   := FALSE;
        stMotionStage.nErrorId := 0;
        bErrorAcknowledge      := FALSE;
    END_IF

    ScaleHomingParams();

    ftHomeVeloFastSetDone   (CLK := fbSetHomeVeloFast.bBusy);
    ftHomeVeloSlowSetDone   (CLK := fbSetHomeVeloSlow.bBusy);
    ftHomeAccSetDone        (CLK := fbSetHomeAcc.bBusy);
    ftHomeOffsSetDone       (CLK := fbSetHomeOffs.bBusy);
    ftReferencingOptSetDone (CLK := fbReferencingOptWrite.bBusy);

    IF tonStartUp.Q OR bForceSequentialSDOs THEN
        CASE nHomingStep OF
            IDLE:
                bHomingParamsSet               := FALSE;
                fbSetHomeVeloFast.bExecute     := FALSE;
                fbSetHomeVeloSlow.bExecute     := FALSE;
                fbSetHomeAcc.bExecute          := FALSE;
                fbSetHomeOffs.bExecute         := FALSE;
                fbReferencingOptWrite.bExecute := FALSE;
                nHomingStep                    := VELO_FAST;

            VELO_FAST:
                IF stMCS2ChanParameter.nHomeVeloFast <> nRecentHomeVeloFast THEN
                    fbSetHomeVeloFast.bExecute := TRUE;
                    IF ftHomeVeloFastSetDone.Q THEN
                        fbSetHomeVeloFast.bExecute := FALSE;
                        IF fbSetHomeVeloFast.bError THEN
                            stMotionStage.bError   := fbSetHomeVeloFast.bError;
                            stMotionStage.nErrorId := fbSetHomeVeloFast.nErrId;
                            nHomingStep            := ERROR;
                        ELSE
                            nRecentHomeVeloFast := stMCS2ChanParameter.nHomeVeloFast;
                            nHomingStep         := VELO_SLOW;
                        END_IF
                    END_IF
                ELSE
                    nHomingStep := VELO_SLOW;
                END_IF

            VELO_SLOW:
                IF stMCS2ChanParameter.nHomeVeloSlow <> nRecentHomeVeloSlow THEN
                    fbSetHomeVeloSlow.bExecute := TRUE;
                    IF ftHomeVeloSlowSetDone.Q THEN
                        fbSetHomeVeloSlow.bExecute := FALSE;
                        IF fbSetHomeVeloSlow.bError THEN
                            stMotionStage.bError   := fbSetHomeVeloSlow.bError;
                            stMotionStage.nErrorId := fbSetHomeVeloSlow.nErrId;
                            nHomingStep            := ERROR;
                        ELSE
                            nRecentHomeVeloSlow := stMCS2ChanParameter.nHomeVeloSlow;
                            nHomingStep         := ACC;
                        END_IF
                    END_IF
                ELSE
                    nHomingStep := ACC;
                END_IF

            ACC:
                IF stMCS2ChanParameter.nHomeAcc <> nRecentHomeAcc THEN
                    fbSetHomeAcc.bExecute := TRUE;
                    IF ftHomeAccSetDone.Q THEN
                        fbSetHomeAcc.bExecute := FALSE;
                        IF fbSetHomeAcc.bError THEN
                            stMotionStage.bError   := fbSetHomeAcc.bError;
                            stMotionStage.nErrorId := fbSetHomeAcc.nErrId;
                            nHomingStep            := ERROR;
                        ELSE
                            nRecentHomeAcc := stMCS2ChanParameter.nHomeAcc;
                            nHomingStep    := OFFSET;
                        END_IF
                    END_IF
                ELSE
                    nHomingStep := OFFSET;
                END_IF

            OFFSET:
                IF stMCS2ChanParameter.nHomeOffset <> nRecentHomeOffset THEN
                    fbSetHomeOffs.bExecute := TRUE;
                    IF ftHomeOffsSetDone.Q THEN
                        fbSetHomeOffs.bExecute := FALSE;
                        IF fbSetHomeOffs.bError THEN
                            stMotionStage.bError   := fbSetHomeOffs.bError;
                            stMotionStage.nErrorId := fbSetHomeOffs.nErrId;
                            nHomingStep            := ERROR;
                        ELSE
                            nRecentHomeOffset := stMCS2ChanParameter.nHomeOffset;
                            nHomingStep       := REF_OPT;
                        END_IF
                    END_IF
                ELSE
                    nHomingStep := REF_OPT;
                END_IF

            REF_OPT:
                IF stMCS2ChanParameter.nReferencingOpt <> nRecentReferencingOpt THEN
                    fbReferencingOptWrite.bExecute := TRUE;
                    IF ftReferencingOptSetDone.Q THEN
                        fbReferencingOptWrite.bExecute := FALSE;
                        IF fbReferencingOptWrite.bError THEN
                            stMotionStage.bError   := fbReferencingOptWrite.bError;
                            stMotionStage.nErrorId := fbReferencingOptWrite.nErrId;
                            nHomingStep            := ERROR;
                        ELSE
                            nRecentReferencingOpt := stMCS2ChanParameter.nReferencingOpt;
                            nHomingStep           := DONE;
                        END_IF
                    END_IF
                ELSE
                    nHomingStep := DONE;
                END_IF

            DONE:
                bHomingParamsSet := TRUE;

            ERROR:
                bHomingParamsSet := FALSE;

            ELSE
                nHomingStep := IDLE;
        END_CASE

    ELSE
        fbSetHomeVeloFast.bExecute     := stMCS2ChanParameter.nHomeVeloFast   <> nRecentHomeVeloFast;
        fbSetHomeVeloSlow.bExecute     := stMCS2ChanParameter.nHomeVeloSlow   <> nRecentHomeVeloSlow;
        fbSetHomeAcc.bExecute          := stMCS2ChanParameter.nHomeAcc        <> nRecentHomeAcc;
        fbSetHomeOffs.bExecute         := stMCS2ChanParameter.nHomeOffset     <> nRecentHomeOffset;
        fbReferencingOptWrite.bExecute := stMCS2ChanParameter.nReferencingOpt <> nRecentReferencingOpt;

        IF ftHomeVeloFastSetDone.Q OR ftHomeVeloSlowSetDone.Q OR ftHomeAccSetDone.Q
            OR ftHomeOffsSetDone.Q OR ftReferencingOptSetDone.Q
        THEN
            IF fbSetHomeVeloFast.bError THEN
                stMotionStage.bError   := fbSetHomeVeloFast.bError;
                stMotionStage.nErrorId := fbSetHomeVeloFast.nErrId;
            ELSIF fbSetHomeVeloSlow.bError THEN
                stMotionStage.bError   := fbSetHomeVeloSlow.bError;
                stMotionStage.nErrorId := fbSetHomeVeloSlow.nErrId;
            ELSIF fbSetHomeAcc.bError THEN
                stMotionStage.bError   := fbSetHomeAcc.bError;
                stMotionStage.nErrorId := fbSetHomeAcc.nErrId;
            ELSIF fbSetHomeOffs.bError THEN
                stMotionStage.bError   := fbSetHomeOffs.bError;
                stMotionStage.nErrorId := fbSetHomeOffs.nErrId;
            ELSIF fbReferencingOptWrite.bError THEN
                stMotionStage.bError   := fbReferencingOptWrite.bError;
                stMotionStage.nErrorId := fbReferencingOptWrite.nErrId;
            ELSE
                nRecentHomeVeloFast   := stMCS2ChanParameter.nHomeVeloFast;
                nRecentHomeVeloSlow   := stMCS2ChanParameter.nHomeVeloSlow;
                nRecentHomeAcc        := stMCS2ChanParameter.nHomeAcc;
                nRecentHomeOffset     := stMCS2ChanParameter.nHomeOffset;
                nRecentReferencingOpt := stMCS2ChanParameter.nReferencingOpt;
                bHomingParamsSet      := TRUE;
            END_IF
            fbSetHomeVeloFast.bExecute     := FALSE;
            fbSetHomeVeloSlow.bExecute     := FALSE;
            fbSetHomeAcc.bExecute          := FALSE;
            fbSetHomeOffs.bExecute         := FALSE;
            fbReferencingOptWrite.bExecute := FALSE;
        END_IF
    END_IF

    fbSetHomeVeloFast(
        sNetId     := stMotionStage.stAxisParameters.sAmsNetId,
        nSlaveAddr := stDS402Drive.nSlaveAddr,
        nIndex     := stMCS2ChanParameter.nChanHomeVeloIdx,
        nSubIndex  := 1,
        pSrcBuf    := ADR(stMCS2ChanParameter.nHomeVeloFast),
        cbBufLen   := SIZEOF(stMCS2ChanParameter.nHomeVeloFast)
    );
    fbSetHomeVeloSlow(
        sNetId     := stMotionStage.stAxisParameters.sAmsNetId,
        nSlaveAddr := stDS402Drive.nSlaveAddr,
        nIndex     := stMCS2ChanParameter.nChanHomeVeloIdx,
        nSubIndex  := 2,
        pSrcBuf    := ADR(stMCS2ChanParameter.nHomeVeloSlow),
        cbBufLen   := SIZEOF(stMCS2ChanParameter.nHomeVeloSlow)
    );
    fbSetHomeAcc(
        sNetId     := stMotionStage.stAxisParameters.sAmsNetId,
        nSlaveAddr := stDS402Drive.nSlaveAddr,
        nIndex     := stMCS2ChanParameter.nChanhomeAccIdx,
        nSubIndex  := 0,
        pSrcBuf    := ADR(stMCS2ChanParameter.nHomeAcc),
        cbBufLen   := SIZEOF(stMCS2ChanParameter.nHomeAcc)
    );
    fbSetHomeOffs(
        sNetId     := stMotionStage.stAxisParameters.sAmsNetId,
        nSlaveAddr := stDS402Drive.nSlaveAddr,
        nIndex     := stMCS2ChanParameter.nChanHomeOffsIdx,
        nSubIndex  := 0,
        pSrcBuf    := ADR(stMCS2ChanParameter.nHomeOffset),
        cbBufLen   := SIZEOF(stMCS2ChanParameter.nHomeOffset)
    );
    fbReferencingOptWrite(
        sNetId     := stMotionStage.stAxisParameters.sAmsNetId,
        nSlaveAddr := stDS402Drive.nSlaveAddr,
        nIndex     := stMCS2ChanParameter.nChanReferencingOptIdx,
        nSubIndex  := 0,
        pSrcBuf    := ADR(stMCS2ChanParameter.nReferencingOpt),
        cbBufLen   := SIZEOF(stMCS2ChanParameter.nReferencingOpt)
    );

    bHomingParamsSet R= fbSetHomeVeloFast.bBusy
                     OR fbSetHomeVeloSlow.bBusy
                     OR fbSetHomeAcc.bBusy
                     OR fbSetHomeOffs.bBusy
                     OR fbReferencingOptWrite.bBusy;
END_IF

(*Scale Home Move parameters*)
METHOD ScaleHomingParams
stMCS2ChanParameter.nHomeVeloFast := LREAL_TO_UDINT(( stMotionStage.stAxisParameters.fRefVeloSearch / MAX( stMotionStage.stAxisParameters.fEncScaleFactorInternal, stMCS2ChanParameter.fScalingFactor)));
stMCS2ChanParameter.nHomeVeloSlow := LREAL_TO_UDINT(( stMotionStage.stAxisParameters.fRefVeloSync / MAX( stMotionStage.stAxisParameters.fEncScaleFactorInternal, stMCS2ChanParameter.fScalingFactor)));
stMCS2ChanParameter.nHomeAcc := LREAL_TO_UDINT((stMCS2ChanParameter.fHomeAcc / MAX( stMotionStage.stAxisParameters.fEncScaleFactorInternal, stMCS2ChanParameter.fScalingFactor)));
stMCS2ChanParameter.nHomeOffset := LREAL_TO_DINT(( stMotionStage.fHomePosition / MAX( stMotionStage.stAxisParameters.fEncScaleFactorInternal, stMCS2ChanParameter.fScalingFactor)));
END_METHOD

END_FUNCTION_BLOCK

// ---- POUs/Motion/DS402/MCS2/FB_WriteStepModeParameters.TcPOU
// Sequential SDOs at startup or when forced; parallel writes otherwise (mirrors Homing Params block).
FUNCTION_BLOCK FB_WriteStepModeParameters
VAR_INPUT
    bEnable : BOOL;
END_VAR
VAR_IN_OUT
    stDS402Drive         : ST_DS402Drive;
    stMotionStage        : ST_MotionStage;
    stMCS2ChanParameter	: ST_MCS2ChanParameter;
END_VAR

VAR_OUTPUT
   bStepModeParamsSet : BOOL;
END_VAR
VAR
    //  Measurements & scaled values
    {attribute 'hide'}
    nScaledFErrWin          : DINT;
    {attribute 'hide'}
    nScalededSteps          : DINT;
    {attribute 'hide'}
    fScalededSteps          : LREAL;
    {attribute 'hide'}
    fMeasuredVelo           : LREAL;
    {attribute 'hide'}
    fMeasuredAcc            : LREAL;
    {attribute 'hide'}
    fParameterValue         : LREAL;
    {attribute 'hide'}
    fMeasuredPos             : LREAL;
    //  Internal numeric parameters
    {attribute 'hide'}
    nScalededStepAmp         : UINT;
    {attribute 'hide'}
    nScaledStepFreq          : UINT;
    // Open Loop Operations
    {attribute 'hide'}
    fbSetSteps          : FB_EcCoESdoWrite;
    {attribute 'hide'}
    fbSetStepFreq       : FB_EcCoESdoWrite;
    {attribute 'hide'}
    fbSetStepAmp        : FB_EcCoESdoWrite;
    {attribute 'hide'}
    nRecentSteps        : DINT;
    {attribute 'hide'}
    nRecentStepAmp      : UINT;
    {attribute 'hide'}
    nRecentStepFreq     : UINT;
    {attribute 'hide'}
    ftStepAmpUpdateDone : F_TRIG;
    {attribute 'hide'}
    ftStepFreqUpdateDone    : F_TRIG;
    {attribute 'hide'}
    ftStepUpdateDone    : F_TRIG;
    tonStartUp : TON;
    nJogParamStep : (IDLE := 0, STEPS := 1, AMP := 2, FREQ := 3, DONE := 10, ERROR := -1) := IDLE;
    bForceSequentialSDOs : BOOL := FALSE;
    bErrorAcknowledge: BOOL;
END_VAR

IF NOT __ISVALIDREF(stDS402Drive)
    OR NOT __ISVALIDREF(stMotionStage)
    OR NOT __ISVALIDREF(stMCS2ChanParameter) THEN
    RETURN;
END_IF

IF bEnable THEN
    tonStartUp(
        IN := bEnable AND NOT bStepModeParamsSet,
        PT := T#5S
    );

    // Reset sequence if startup timer hasn't fired and not forcing sequential SDOs
    IF NOT tonStartUp.Q AND nJogParamStep <> IDLE AND NOT bForceSequentialSDOs THEN
        nJogParamStep := IDLE;
    END_IF

    // Acknowledge error and restart sequence
    IF nJogParamStep = ERROR AND bErrorAcknowledge THEN
        nJogParamStep          := IDLE;
        stMotionStage.bError   := FALSE;
        stMotionStage.nErrorId := 0;
    END_IF

    ScaleStepModeParams();

    ftStepUpdateDone    (CLK := fbSetSteps.bBusy);
    ftStepAmpUpdateDone (CLK := fbSetStepAmp.bBusy);
    ftStepFreqUpdateDone(CLK := fbSetStepFreq.bBusy);

    IF tonStartUp.Q OR bForceSequentialSDOs THEN
        CASE nJogParamStep OF
            IDLE:
                bStepModeParamsSet      := FALSE;
                fbSetSteps.bExecute     := FALSE;
                fbSetStepAmp.bExecute   := FALSE;
                fbSetStepFreq.bExecute  := FALSE;
                nJogParamStep           := STEPS;

            STEPS:
                IF nScalededSteps <> nRecentSteps THEN
                    fbSetSteps.bExecute := TRUE;
                    IF ftStepUpdateDone.Q THEN
                        IF fbSetSteps.bError THEN
                            stMotionStage.bError   := fbSetSteps.bError;
                            stMotionStage.nErrorId := fbSetSteps.nErrId;
                            nJogParamStep          := ERROR;
                        ELSE
                            nRecentSteps        := nScalededSteps;
                            fbSetSteps.bExecute := FALSE;
                            nJogParamStep       := AMP;
                        END_IF
                    END_IF
                ELSE
                    nJogParamStep := AMP;
                END_IF

            AMP:
                IF nScalededStepAmp <> nRecentStepAmp THEN
                    fbSetStepAmp.bExecute := TRUE;
                    IF ftStepAmpUpdateDone.Q THEN
                        IF fbSetStepAmp.bError THEN
                            stMotionStage.bError   := fbSetStepAmp.bError;
                            stMotionStage.nErrorId := fbSetStepAmp.nErrId;
                            nJogParamStep          := ERROR;
                        ELSE
                            nRecentStepAmp          := nScalededStepAmp;
                            fbSetStepAmp.bExecute   := FALSE;
                            nJogParamStep           := FREQ;
                        END_IF
                    END_IF
                ELSE
                    nJogParamStep := FREQ;
                END_IF

            FREQ:
                IF nScaledStepFreq <> nRecentStepFreq THEN
                    fbSetStepFreq.bExecute := TRUE;
                    IF ftStepFreqUpdateDone.Q THEN
                        IF fbSetStepFreq.bError THEN
                            stMotionStage.bError   := fbSetStepFreq.bError;
                            stMotionStage.nErrorId := fbSetStepFreq.nErrId;
                            nJogParamStep          := ERROR;
                        ELSE
                            nRecentStepFreq         := nScaledStepFreq;
                            fbSetStepFreq.bExecute  := FALSE;
                            nJogParamStep           := DONE;
                        END_IF
                    END_IF
                ELSE
                    nJogParamStep := DONE;
                END_IF

            DONE:
                bStepModeParamsSet := TRUE;

            ERROR:
                bStepModeParamsSet := FALSE;

            ELSE
                nJogParamStep := IDLE;
        END_CASE

    ELSE
        // Parallel SDO mode — fire all three simultaneously
        fbSetSteps.bExecute    := nScalededSteps   <> nRecentSteps;
        fbSetStepAmp.bExecute  := nScalededStepAmp <> nRecentStepAmp;
        fbSetStepFreq.bExecute := nScaledStepFreq  <> nRecentStepFreq;

        IF ftStepUpdateDone.Q OR ftStepAmpUpdateDone.Q OR ftStepFreqUpdateDone.Q THEN
            IF fbSetSteps.bError THEN
                stMotionStage.bError   := fbSetSteps.bError;
                stMotionStage.nErrorId := fbSetSteps.nErrId;
            ELSIF fbSetStepAmp.bError THEN
                stMotionStage.bError   := fbSetStepAmp.bError;
                stMotionStage.nErrorId := fbSetStepAmp.nErrId;
            ELSIF fbSetStepFreq.bError THEN
                stMotionStage.bError   := fbSetStepFreq.bError;
                stMotionStage.nErrorId := fbSetStepFreq.nErrId;
            ELSE
                nRecentSteps       := nScalededSteps;
                nRecentStepAmp     := nScalededStepAmp;
                nRecentStepFreq    := nScaledStepFreq;
                bStepModeParamsSet := TRUE;
            END_IF
            fbSetSteps.bExecute    := FALSE;
            fbSetStepAmp.bExecute  := FALSE;
            fbSetStepFreq.bExecute := FALSE;
        END_IF
    END_IF

    fbSetSteps(
        sNetId     := stMotionStage.stAxisParameters.sAmsNetId,
        nSlaveAddr := stDS402Drive.nSlaveAddr,
        nIndex     := stMCS2ChanParameter.nChanStepIdx,
        nSubIndex  := 0,
        pSrcBuf    := ADR(nScalededSteps),
        cbBufLen   := SIZEOF(stMCS2ChanParameter.nChanStep)
    );
    fbSetStepAmp(
        sNetId     := stMotionStage.stAxisParameters.sAmsNetId,
        nSlaveAddr := stDS402Drive.nSlaveAddr,
        nIndex     := stMCS2ChanParameter.nChanStepAmpIdx,
        nSubIndex  := 0,
        pSrcBuf    := ADR(nScalededStepAmp),
        cbBufLen   := SIZEOF(stMCS2ChanParameter.nChanStepAmp)
    );
    fbSetStepFreq(
        sNetId     := stMotionStage.stAxisParameters.sAmsNetId,
        nSlaveAddr := stDS402Drive.nSlaveAddr,
        nIndex     := stMCS2ChanParameter.nChanStepFreqIdx,
        nSubIndex  := 0,
        pSrcBuf    := ADR(nScaledStepFreq),
        cbBufLen   := SIZEOF(stMCS2ChanParameter.nChanStepFreq)
    );

    bStepModeParamsSet R= fbSetSteps.bBusy
                       OR fbSetStepAmp.bBusy
                       OR fbSetStepFreq.bBusy;
END_IF

(*Scaled Open Loop Step mode motion parameters*)
METHOD ScaleStepModeParams
VAR_INPUT
END_VAR
//827.31x-837.63
nScalededSteps:=LIMIT(-1000, stMCS2ChanParameter.nChanStep, 1000);
nScalededStepAmp:=REAL_TO_UINT(LIMIT(50, stMCS2ChanParameter.nChanStepAmp, 100) * 655.35);
nScaledStepFreq:=REAL_TO_UINT(LIMIT(500, stMCS2ChanParameter.nChanStepFreq, 1000.0));
END_METHOD

END_FUNCTION_BLOCK

